REGION Network 115: NG 1 Door NOT Closed
   RUNG wire#powerrail
      Contact( "AlwaysTRUE" )
      Contact( "Station_Sys".Auto.Mode )
      I_Contact( "oE-NG-01SafetyGate" )
      Coil( "ST10_DeviceError"."E".NG_1."NG 1 DoorOpen" )
   END_RUNG
   // the same network as SCL:
   "ST10_DeviceError"."E".NG_1."NG 1 DoorOpen" := "AlwaysTRUE" AND "Station_Sys".Auto.Mode AND NOT "oE-NG-01SafetyGate";
END_REGION

REGION Network 116: E NG_2
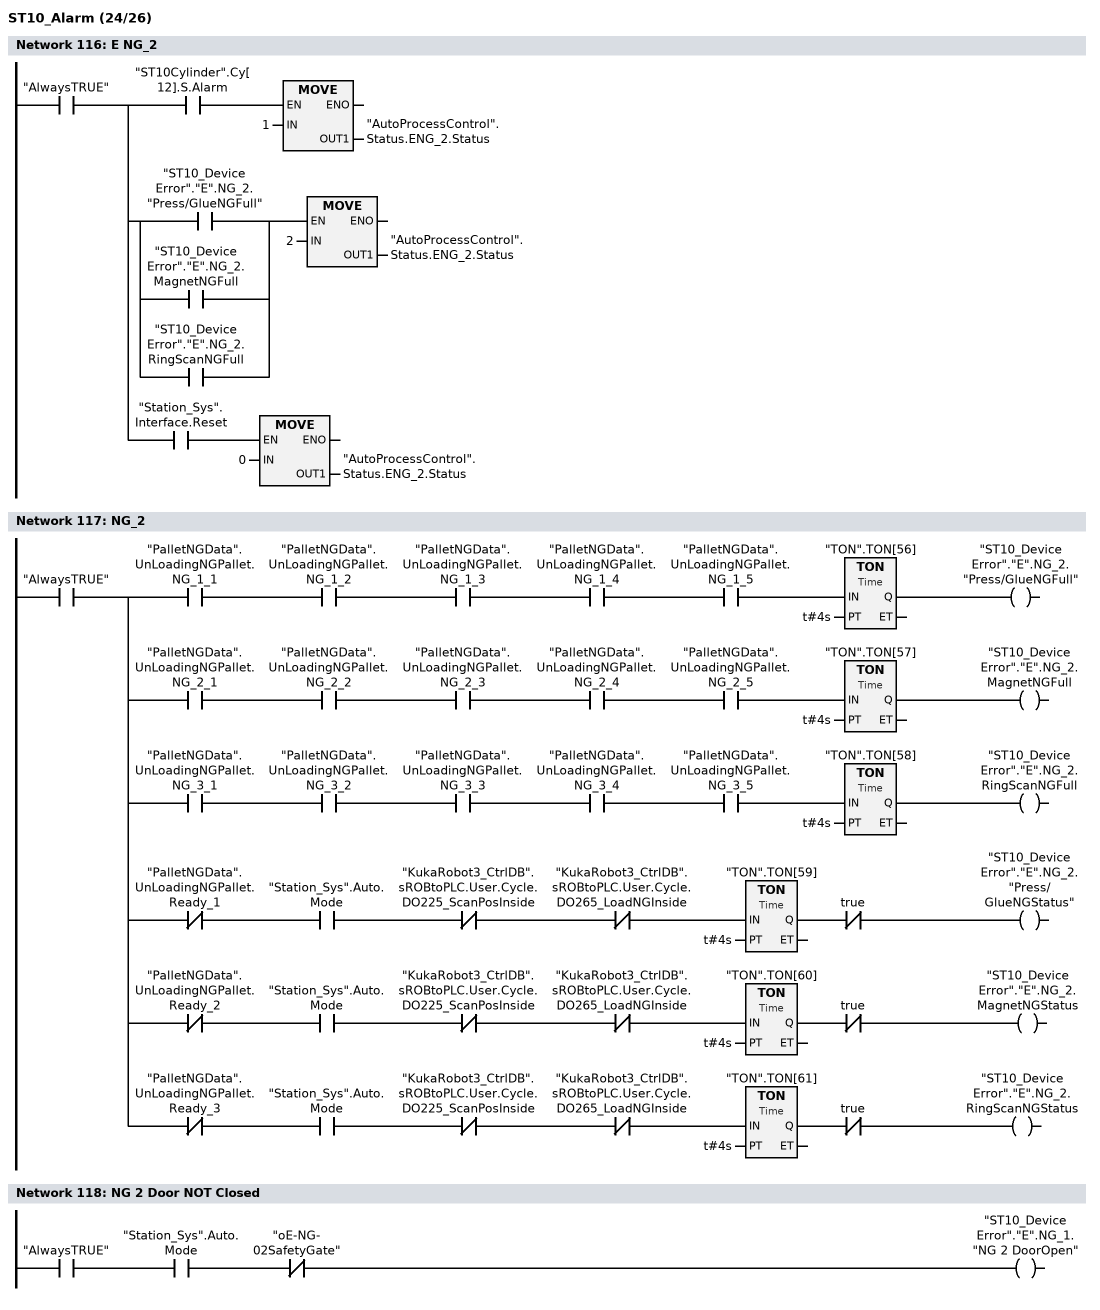
   RUNG wire#powerrail
      Contact( "AlwaysTRUE" )
      wire#w1
      Contact( "ST10Cylinder".Cy[12].S.Alarm )
      Move(in := 1, out1 => "AutoProcessControl".Status.ENG_2.Status)
   END_RUNG
   RUNG wire#w1
      Contact( "ST10_DeviceError"."E".NG_2."Press/GlueNGFull" )
      wire#w2
      Move(in := 2, out1 => "AutoProcessControl".Status.ENG_2.Status)
   END_RUNG
   RUNG wire#w1
      Contact( "ST10_DeviceError"."E".NG_2.MagnetNGFull )
   END_RUNG wire#w2
   RUNG wire#w1
      Contact( "ST10_DeviceError"."E".NG_2.RingScanNGFull )
   END_RUNG wire#w2
   RUNG wire#w1
      Contact( "Station_Sys".Interface.Reset )
      Move(in := 0, out1 => "AutoProcessControl".Status.ENG_2.Status)
   END_RUNG
   // the same network as SCL:
   IF "AlwaysTRUE" AND "ST10Cylinder".Cy[12].S.Alarm THEN
       "AutoProcessControl".Status.ENG_2.Status := 1;
   END_IF;
   IF "AlwaysTRUE" AND ("ST10_DeviceError"."E".NG_2."Press/GlueNGFull" OR "ST10_DeviceError"."E".NG_2.MagnetNGFull OR "ST10_DeviceError"."E".NG_2.RingScanNGFull) THEN
       "AutoProcessControl".Status.ENG_2.Status := 2;
   END_IF;
   IF "AlwaysTRUE" AND "Station_Sys".Interface.Reset THEN
       "AutoProcessControl".Status.ENG_2.Status := 0;
   END_IF;
END_REGION

REGION Network 117: NG_2
   RUNG wire#powerrail
      Contact( "AlwaysTRUE" )
      wire#w1
      Contact( "PalletNGData".UnLoadingNGPallet.NG_1_1 )
      Contact( "PalletNGData".UnLoadingNGPallet.NG_1_2 )
      Contact( "PalletNGData".UnLoadingNGPallet.NG_1_3 )
      Contact( "PalletNGData".UnLoadingNGPallet.NG_1_4 )
      Contact( "PalletNGData".UnLoadingNGPallet.NG_1_5 )
      { S7_Templates := "time_type := Time" } "TON".TON[56].TON(pt := t#4s, et =>)
      Coil( "ST10_DeviceError"."E".NG_2."Press/GlueNGFull" )
   END_RUNG
   RUNG wire#w1
      Contact( "PalletNGData".UnLoadingNGPallet.NG_2_1 )
      Contact( "PalletNGData".UnLoadingNGPallet.NG_2_2 )
      Contact( "PalletNGData".UnLoadingNGPallet.NG_2_3 )
      Contact( "PalletNGData".UnLoadingNGPallet.NG_2_4 )
      Contact( "PalletNGData".UnLoadingNGPallet.NG_2_5 )
      { S7_Templates := "time_type := Time" } "TON".TON[57].TON(pt := t#4s, et =>)
      Coil( "ST10_DeviceError"."E".NG_2.MagnetNGFull )
   END_RUNG
   RUNG wire#w1
      Contact( "PalletNGData".UnLoadingNGPallet.NG_3_1 )
      Contact( "PalletNGData".UnLoadingNGPallet.NG_3_2 )
      Contact( "PalletNGData".UnLoadingNGPallet.NG_3_3 )
      Contact( "PalletNGData".UnLoadingNGPallet.NG_3_4 )
      Contact( "PalletNGData".UnLoadingNGPallet.NG_3_5 )
      { S7_Templates := "time_type := Time" } "TON".TON[58].TON(pt := t#4s, et =>)
      Coil( "ST10_DeviceError"."E".NG_2.RingScanNGFull )
   END_RUNG
   RUNG wire#w1
      I_Contact( "PalletNGData".UnLoadingNGPallet.Ready_1 )
      Contact( "Station_Sys".Auto.Mode )
      I_Contact( "KukaRobot3_CtrlDB".sROBtoPLC.User.Cycle.DO225_ScanPosInside )
      I_Contact( "KukaRobot3_CtrlDB".sROBtoPLC.User.Cycle.DO265_LoadNGInside )
      { S7_Templates := "time_type := Time" } "TON".TON[59].TON(pt := t#4s, et =>)
      I_Contact( true )
      Coil( "ST10_DeviceError"."E".NG_2."Press/GlueNGStatus" )
   END_RUNG
   RUNG wire#w1
      I_Contact( "PalletNGData".UnLoadingNGPallet.Ready_2 )
      Contact( "Station_Sys".Auto.Mode )
      I_Contact( "KukaRobot3_CtrlDB".sROBtoPLC.User.Cycle.DO225_ScanPosInside )
      I_Contact( "KukaRobot3_CtrlDB".sROBtoPLC.User.Cycle.DO265_LoadNGInside )
      { S7_Templates := "time_type := Time" } "TON".TON[60].TON(pt := t#4s, et =>)
      I_Contact( true )
      Coil( "ST10_DeviceError"."E".NG_2.MagnetNGStatus )
   END_RUNG
   RUNG wire#w1
      I_Contact( "PalletNGData".UnLoadingNGPallet.Ready_3 )
      Contact( "Station_Sys".Auto.Mode )
      I_Contact( "KukaRobot3_CtrlDB".sROBtoPLC.User.Cycle.DO225_ScanPosInside )
      I_Contact( "KukaRobot3_CtrlDB".sROBtoPLC.User.Cycle.DO265_LoadNGInside )
      { S7_Templates := "time_type := Time" } "TON".TON[61].TON(pt := t#4s, et =>)
      I_Contact( true )
      Coil( "ST10_DeviceError"."E".NG_2.RingScanNGStatus )
   END_RUNG
   // the same network as SCL:
   "TON".TON[56].TON(IN := "AlwaysTRUE" AND "PalletNGData".UnLoadingNGPallet.NG_1_1 AND "PalletNGData".UnLoadingNGPallet.NG_1_2 AND "PalletNGData".UnLoadingNGPallet.NG_1_3 AND "PalletNGData".UnLoadingNGPallet.NG_1_4 AND "PalletNGData".UnLoadingNGPallet.NG_1_5,
                     PT := t#4s);
   "ST10_DeviceError"."E".NG_2."Press/GlueNGFull" := "TON".TON[56].Q;
   "TON".TON[57].TON(IN := "AlwaysTRUE" AND "PalletNGData".UnLoadingNGPallet.NG_2_1 AND "PalletNGData".UnLoadingNGPallet.NG_2_2 AND "PalletNGData".UnLoadingNGPallet.NG_2_3 AND "PalletNGData".UnLoadingNGPallet.NG_2_4 AND "PalletNGData".UnLoadingNGPallet.NG_2_5,
                     PT := t#4s);
   "ST10_DeviceError"."E".NG_2.MagnetNGFull := "TON".TON[57].Q;
   "TON".TON[58].TON(IN := "AlwaysTRUE" AND "PalletNGData".UnLoadingNGPallet.NG_3_1 AND "PalletNGData".UnLoadingNGPallet.NG_3_2 AND "PalletNGData".UnLoadingNGPallet.NG_3_3 AND "PalletNGData".UnLoadingNGPallet.NG_3_4 AND "PalletNGData".UnLoadingNGPallet.NG_3_5,
                     PT := t#4s);
   "ST10_DeviceError"."E".NG_2.RingScanNGFull := "TON".TON[58].Q;
   "TON".TON[59].TON(IN := "AlwaysTRUE" AND NOT "PalletNGData".UnLoadingNGPallet.Ready_1 AND "Station_Sys".Auto.Mode AND NOT "KukaRobot3_CtrlDB".sROBtoPLC.User.Cycle.DO225_ScanPosInside AND NOT "KukaRobot3_CtrlDB".sROBtoPLC.User.Cycle.DO265_LoadNGInside,
                     PT := t#4s);
   "ST10_DeviceError"."E".NG_2."Press/GlueNGStatus" := "TON".TON[59].Q AND NOT true;
   "TON".TON[60].TON(IN := "AlwaysTRUE" AND NOT "PalletNGData".UnLoadingNGPallet.Ready_2 AND "Station_Sys".Auto.Mode AND NOT "KukaRobot3_CtrlDB".sROBtoPLC.User.Cycle.DO225_ScanPosInside AND NOT "KukaRobot3_CtrlDB".sROBtoPLC.User.Cycle.DO265_LoadNGInside,
                     PT := t#4s);
   "ST10_DeviceError"."E".NG_2.MagnetNGStatus := "TON".TON[60].Q AND NOT true;
   "TON".TON[61].TON(IN := "AlwaysTRUE" AND NOT "PalletNGData".UnLoadingNGPallet.Ready_3 AND "Station_Sys".Auto.Mode AND NOT "KukaRobot3_CtrlDB".sROBtoPLC.User.Cycle.DO225_ScanPosInside AND NOT "KukaRobot3_CtrlDB".sROBtoPLC.User.Cycle.DO265_LoadNGInside,
                     PT := t#4s);
   "ST10_DeviceError"."E".NG_2.RingScanNGStatus := "TON".TON[61].Q AND NOT true;
END_REGION

REGION Network 118: NG 2 Door NOT Closed
   RUNG wire#powerrail
      Contact( "AlwaysTRUE" )
      Contact( "Station_Sys".Auto.Mode )
      I_Contact( "oE-NG-02SafetyGate" )
      Coil( "ST10_DeviceError"."E".NG_1."NG 2 DoorOpen" )
   END_RUNG
   // the same network as SCL:
   "ST10_DeviceError"."E".NG_1."NG 2 DoorOpen" := "AlwaysTRUE" AND "Station_Sys".Auto.Mode AND NOT "oE-NG-02SafetyGate";
END_REGION

REGION Network 119: Press1
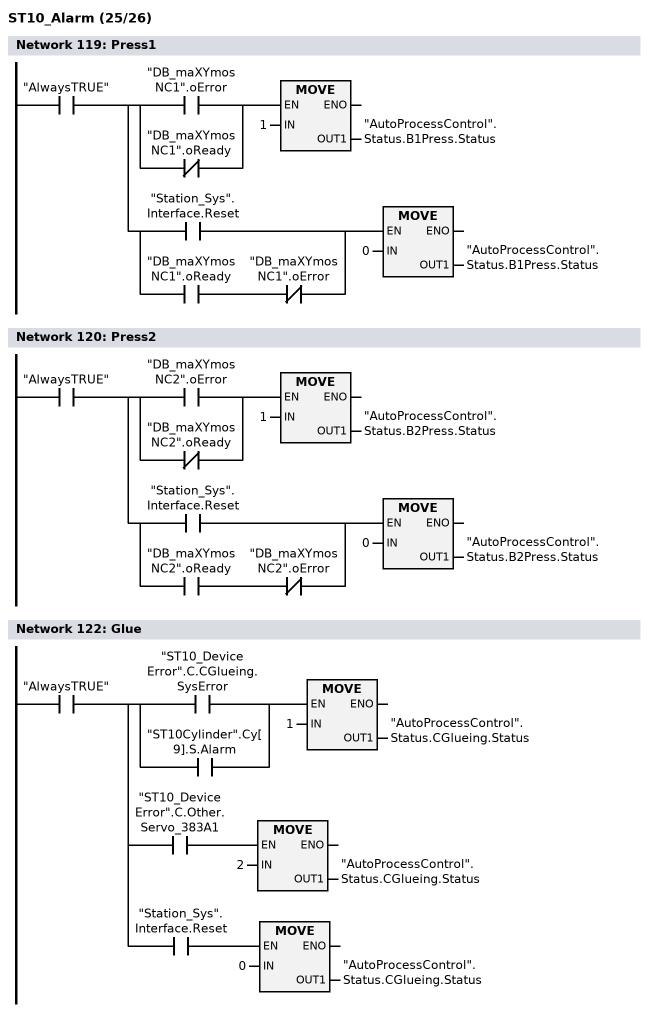
   RUNG wire#powerrail
      Contact( "AlwaysTRUE" )
      wire#w1
      Contact( "DB_maXYmosNC1".oError )
      wire#w2
      Move(in := 1, out1 => "AutoProcessControl".Status.B1Press.Status)
   END_RUNG
   RUNG wire#w1
      I_Contact( "DB_maXYmosNC1".oReady )
   END_RUNG wire#w2
   RUNG wire#w1
      Contact( "Station_Sys".Interface.Reset )
      wire#w3
      Move(in := 0, out1 => "AutoProcessControl".Status.B1Press.Status)
   END_RUNG
   RUNG wire#w1
      Contact( "DB_maXYmosNC1".oReady )
      I_Contact( "DB_maXYmosNC1".oError )
   END_RUNG wire#w3
   // the same network as SCL:
   IF "AlwaysTRUE" AND ("DB_maXYmosNC1".oError OR NOT "DB_maXYmosNC1".oReady) THEN
       "AutoProcessControl".Status.B1Press.Status := 1;
   END_IF;
   IF "AlwaysTRUE" AND ("Station_Sys".Interface.Reset OR ("DB_maXYmosNC1".oReady AND NOT "DB_maXYmosNC1".oError)) THEN
       "AutoProcessControl".Status.B1Press.Status := 0;
   END_IF;
END_REGION

REGION Network 120: Press2
   RUNG wire#powerrail
      Contact( "AlwaysTRUE" )
      wire#w1
      Contact( "DB_maXYmosNC2".oError )
      wire#w2
      Move(in := 1, out1 => "AutoProcessControl".Status.B2Press.Status)
   END_RUNG
   RUNG wire#w1
      I_Contact( "DB_maXYmosNC2".oReady )
   END_RUNG wire#w2
   RUNG wire#w1
      Contact( "Station_Sys".Interface.Reset )
      wire#w3
      Move(in := 0, out1 => "AutoProcessControl".Status.B2Press.Status)
   END_RUNG
   RUNG wire#w1
      Contact( "DB_maXYmosNC2".oReady )
      I_Contact( "DB_maXYmosNC2".oError )
   END_RUNG wire#w3
   // the same network as SCL:
   IF "AlwaysTRUE" AND ("DB_maXYmosNC2".oError OR NOT "DB_maXYmosNC2".oReady) THEN
       "AutoProcessControl".Status.B2Press.Status := 1;
   END_IF;
   IF "AlwaysTRUE" AND ("Station_Sys".Interface.Reset OR ("DB_maXYmosNC2".oReady AND NOT "DB_maXYmosNC2".oError)) THEN
       "AutoProcessControl".Status.B2Press.Status := 0;
   END_IF;
END_REGION

REGION Network 121: ******************** Glue ********************
END_REGION

REGION Network 122: Glue
   RUNG wire#powerrail
      Contact( "AlwaysTRUE" )
      wire#w1
      Contact( "ST10_DeviceError".C.CGlueing.SysError )
      wire#w2
      Move(in := 1, out1 => "AutoProcessControl".Status.CGlueing.Status)
   END_RUNG
   RUNG wire#w1
      Contact( "ST10Cylinder".Cy[9].S.Alarm )
   END_RUNG wire#w2
   RUNG wire#w1
      Contact( "ST10_DeviceError".C.Other.Servo_383A1 )
      Move(in := 2, out1 => "AutoProcessControl".Status.CGlueing.Status)
   END_RUNG
   RUNG wire#w1
      Contact( "Station_Sys".Interface.Reset )
      Move(in := 0, out1 => "AutoProcessControl".Status.CGlueing.Status)
   END_RUNG
   // the same network as SCL:
   IF "AlwaysTRUE" AND ("ST10_DeviceError".C.CGlueing.SysError OR "ST10Cylinder".Cy[9].S.Alarm) THEN
       "AutoProcessControl".Status.CGlueing.Status := 1;
   END_IF;
   IF "AlwaysTRUE" AND "ST10_DeviceError".C.Other.Servo_383A1 THEN
       "AutoProcessControl".Status.CGlueing.Status := 2;
   END_IF;
   IF "AlwaysTRUE" AND "Station_Sys".Interface.Reset THEN
       "AutoProcessControl".Status.CGlueing.Status := 0;
   END_IF;
END_REGION

REGION Network 123: A1 Table
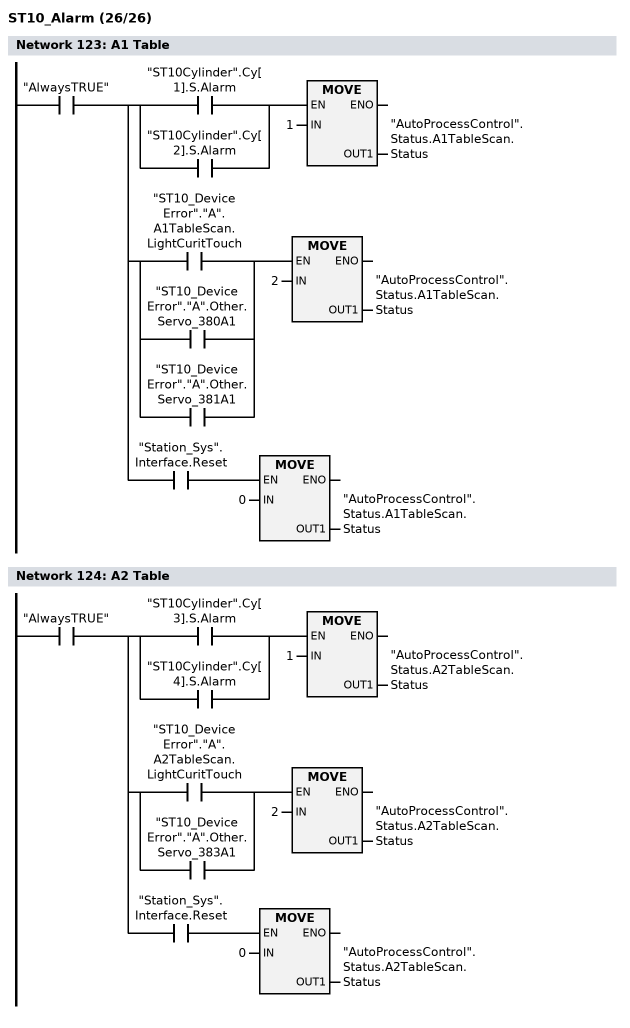
   RUNG wire#powerrail
      Contact( "AlwaysTRUE" )
      wire#w1
      Contact( "ST10Cylinder".Cy[1].S.Alarm )
      wire#w2
      Move(in := 1, out1 => "AutoProcessControl".Status.A1TableScan.Status)
   END_RUNG
   RUNG wire#w1
      Contact( "ST10Cylinder".Cy[2].S.Alarm )
   END_RUNG wire#w2
   RUNG wire#w1
      Contact( "ST10_DeviceError"."A".A1TableScan.LightCuritTouch )
      wire#w3
      Move(in := 2, out1 => "AutoProcessControl".Status.A1TableScan.Status)
   END_RUNG
   RUNG wire#w1
      Contact( "ST10_DeviceError"."A".Other.Servo_380A1 )
   END_RUNG wire#w3
   RUNG wire#w1
      Contact( "ST10_DeviceError"."A".Other.Servo_381A1 )
   END_RUNG wire#w3
   RUNG wire#w1
      Contact( "Station_Sys".Interface.Reset )
      Move(in := 0, out1 => "AutoProcessControl".Status.A1TableScan.Status)
   END_RUNG
   // the same network as SCL:
   IF "AlwaysTRUE" AND ("ST10Cylinder".Cy[1].S.Alarm OR "ST10Cylinder".Cy[2].S.Alarm) THEN
       "AutoProcessControl".Status.A1TableScan.Status := 1;
   END_IF;
   IF "AlwaysTRUE" AND ("ST10_DeviceError"."A".A1TableScan.LightCuritTouch OR "ST10_DeviceError"."A".Other.Servo_380A1 OR "ST10_DeviceError"."A".Other.Servo_381A1) THEN
       "AutoProcessControl".Status.A1TableScan.Status := 2;
   END_IF;
   IF "AlwaysTRUE" AND "Station_Sys".Interface.Reset THEN
       "AutoProcessControl".Status.A1TableScan.Status := 0;
   END_IF;
END_REGION

REGION Network 124: A2 Table
   RUNG wire#powerrail
      Contact( "AlwaysTRUE" )
      wire#w1
      Contact( "ST10Cylinder".Cy[3].S.Alarm )
      wire#w2
      Move(in := 1, out1 => "AutoProcessControl".Status.A2TableScan.Status)
   END_RUNG
   RUNG wire#w1
      Contact( "ST10Cylinder".Cy[4].S.Alarm )
   END_RUNG wire#w2
   RUNG wire#w1
      Contact( "ST10_DeviceError"."A".A2TableScan.LightCuritTouch )
      wire#w3
      Move(in := 2, out1 => "AutoProcessControl".Status.A2TableScan.Status)
   END_RUNG
   RUNG wire#w1
      Contact( "ST10_DeviceError"."A".Other.Servo_383A1 )
   END_RUNG wire#w3
   RUNG wire#w1
      Contact( "Station_Sys".Interface.Reset )
      Move(in := 0, out1 => "AutoProcessControl".Status.A2TableScan.Status)
   END_RUNG
   // the same network as SCL:
   IF "AlwaysTRUE" AND ("ST10Cylinder".Cy[3].S.Alarm OR "ST10Cylinder".Cy[4].S.Alarm) THEN
       "AutoProcessControl".Status.A2TableScan.Status := 1;
   END_IF;
   IF "AlwaysTRUE" AND ("ST10_DeviceError"."A".A2TableScan.LightCuritTouch OR "ST10_DeviceError"."A".Other.Servo_383A1) THEN
       "AutoProcessControl".Status.A2TableScan.Status := 2;
   END_IF;
   IF "AlwaysTRUE" AND "Station_Sys".Interface.Reset THEN
       "AutoProcessControl".Status.A2TableScan.Status := 0;
   END_IF;
END_REGION
END_FUNCTION

FUNCTION "ST10Cyl_interface11-20" : Void   // FC1021, LAD
{ S7_Optimized_Access := 'FALSE' }
// stored: AutoNumber false, SetENOAutomatically false
   VAR_INPUT
      AlwaysON : Bool;
      E_stop : Bool;
   END_VAR
   VAR_TEMP
      tTest : Bool;
   END_VAR
BEGIN

REGION Network 1 (SCL): Cylinder 11-20 IO Interface (SCL)

   //Cylinder11 IO   E-NG-01NGLocationCylinder
   //Input
   "ST10Cylinder".Cy[11].In.WorkPositionSensor := "iE-NG-01NGLocationCylinderInWP";
   "ST10Cylinder".Cy[11].In.HomePositionSensor := "iE-NG-01NGLocationCylinderInHP";
   //Output
   "oE-NG-01NGLocationCylinderToWP" := "ST10Cylinder".Cy[11].Out.GoWorkPosition;
   "oE-NG-01NGLocationCylinderToHP" := "ST10Cylinder".Cy[11].Out.GoHomePosition;

   //Cylinder12 IO  E-NG-02NGLocationCylinder
   //Input
   "ST10Cylinder".Cy[12].In.WorkPositionSensor := "iE-NG-02NGLocationCylinderInWP";
   "ST10Cylinder".Cy[12].In.HomePositionSensor := "iE-NG-02NGLocationCylinderInHP";
   //Output
   "oE-NG-02NGLocationCylinderToWP" := "ST10Cylinder".Cy[12].Out.GoWorkPosition;
   "oE-NG-02NGLocationCylinderToHP" := "ST10Cylinder".Cy[12].Out.GoHomePosition;

   //Cylinder13 IO  F-ROOBT1Gripper1Cylinder
   //Input
   "KukaRobot1_CtrlDB".sPLCtoROB.User.Gripper.DI129_Grip1WP:="ST10Cylinder".Cy[13].In.WorkPositionSensor := "iF-ROOBT1Gripper1CylinderInWP" ;
   "KukaRobot1_CtrlDB".sPLCtoROB.User.Gripper.DI130_Grip1HP := "ST10Cylinder".Cy[13].In.HomePositionSensor := "iF-ROOBT1Gripper1CylinderInHP" ;//"TON".TON[0].Q;

   IF  NOT "Robot_DB".Control.Robot1GripControl THEN
       //Output
       "oF-ROOBT1Gripper1CylinderToWP" := "KukaRobot1_CtrlDB".sROBtoPLC.User.Gripper.DO129_Grip1GoWork;
       "oF-ROOBT1Gripper1CylinderToHP" := "KukaRobot1_CtrlDB".sROBtoPLC.User.Gripper.DO130_Grip1GoHome;
   ELSE
       //Output
       "oF-ROOBT1Gripper1CylinderToWP" := "ST10Cylinder".Cy[13].Out.GoWorkPosition;
       "oF-ROOBT1Gripper1CylinderToHP" := "ST10Cylinder".Cy[13].Out.GoHomePosition;
   END_IF;
   "TON".TON[0](IN:="oF-ROOBT1Gripper1CylinderToHP" AND NOT"iF-ROOBT1Gripper1CylinderInWP",PT:=T#500MS);


   //Cylinder14 IO  F-ROOBT1Gripper2Cylinder
   //Input
   "KukaRobot1_CtrlDB".sPLCtoROB.User.Gripper.DI131_Grip2WP:="ST10Cylinder".Cy[14].In.WorkPositionSensor := "iF-ROOBT1Gripper2CylinderInWP";
   "KukaRobot1_CtrlDB".sPLCtoROB.User.Gripper.DI132_Grip2HP:="ST10Cylinder".Cy[14].In.HomePositionSensor := "iF-ROOBT1Gripper2CylinderInHP";

   IF NOT "Robot_DB".Control.Robot1GripControl THEN
       //Output
       "oF-ROOBT1Gripper2CylinderToWP" :="ST10Cylinder".Cy[14].Inout.AutoGoWork:="KukaRobot1_CtrlDB".sROBtoPLC.User.Gripper.DO131_Grip2GoWork;
       "oF-ROOBT1Gripper2CylinderToHP" :="ST10Cylinder".Cy[14].Inout.AutoGoHome:="KukaRobot1_CtrlDB".sROBtoPLC.User.Gripper.DO132_Grip2GoHome;
   ELSE
       //Output
       "oF-ROOBT1Gripper2CylinderToWP" := "ST10Cylinder".Cy[14].Out.GoWorkPosition;
       "oF-ROOBT1Gripper2CylinderToHP" := "ST10Cylinder".Cy[14].Out.GoHomePosition;
   END_IF;


   //Cylinder15 IO  F-ROOBT2Gripper1Cylinder
   //Input
   "KukaRobot2_CtrlDB".sPLCtoROB.User.Gripper.DI129_Grip1WP:="ST10Cylinder".Cy[15].In.WorkPositionSensor := "iF-ROOBT2Gripper1CylinderInWP";
   "KukaRobot2_CtrlDB".sPLCtoROB.User.Gripper.DI130_Grip1HP := "ST10Cylinder".Cy[15].In.HomePositionSensor :="iF-ROOBT2Gripper1CylinderInHP";

   IF NOT "Robot_DB".Control.Robot2GripControl THEN
       //Output
       "oF-ROOBT2Gripper1CylinderToWP" :="ST10Cylinder".Cy[15].Inout.AutoGoWork:="KukaRobot2_CtrlDB".sROBtoPLC.User.Gripper.DO129_Grip1GoWork;
       "oF-ROOBT2Gripper1CylinderToHP" :="ST10Cylinder".Cy[15].Inout.AutoGoHome:="KukaRobot2_CtrlDB".sROBtoPLC.User.Gripper.DO130_Grip1GoHome;
   ELSE
       //Output
       "oF-ROOBT2Gripper1CylinderToWP" := "ST10Cylinder".Cy[15].Out.GoWorkPosition;
       "oF-ROOBT2Gripper1CylinderToHP" := "ST10Cylinder".Cy[15].Out.GoHomePosition;
   END_IF;



   //Cylinder16 IO  F-ROOBT2Gripper2Cylinder
   //Input
   "KukaRobot2_CtrlDB".sPLCtoROB.User.Gripper.DI131_Grip2WP:="ST10Cylinder".Cy[16].In.WorkPositionSensor := "iF-ROOBT2Gripper2CylinderInWP";
   "KukaRobot2_CtrlDB".sPLCtoROB.User.Gripper.DI132_Grip2HP:="ST10Cylinder".Cy[16].In.HomePositionSensor := "iF-ROOBT2Gripper2CylinderInHP";

   IF NOT "Robot_DB".Control.Robot2GripControl THEN
       //Output
       "oF-ROOBT2Gripper2CylinderToWP" :="ST10Cylinder".Cy[16].Inout.AutoGoWork:= "KukaRobot2_CtrlDB".sROBtoPLC.User.Gripper.DO131_Grip2GoWork;
       "oF-ROOBT2Gripper2CylinderToHP" :="ST10Cylinder".Cy[16].Inout.AutoGoHome:= "KukaRobot2_CtrlDB".sROBtoPLC.User.Gripper.DO132_Grip2GoHome;
   ELSE
       //Output
       "oF-ROOBT2Gripper2CylinderToWP" := "ST10Cylinder".Cy[16].Out.GoWorkPosition;
       "oF-ROOBT2Gripper2CylinderToHP" := "ST10Cylinder".Cy[16].Out.GoHomePosition;
   END_IF;

   //Cylinder17 IO  F-ROOBT3Gripper1Cylinder
   //Input
   "KukaRobot3_CtrlDB".sPLCtoROB.User.Gripper.DI129_Grip1WP:="ST10Cylinder".Cy[17].In.WorkPositionSensor := "iF-ROOBT3Gripper1CylinderInWP";
   "KukaRobot3_CtrlDB".sPLCtoROB.User.Gripper.DI130_Grip1HP:="ST10Cylinder".Cy[17].In.HomePositionSensor := "iF-ROOBT3Gripper1CylinderInHP";

   IF NOT "Robot_DB".Control.Robot3GripControl THEN
       //Output
       "oF-ROOBT3Gripper1CylinderToWP" :="ST10Cylinder".Cy[17].Inout.AutoGoWork:="KukaRobot3_CtrlDB".sROBtoPLC.User.Gripper.DO129_Grip1GoWork;
       "oF-ROOBT3Gripper1CylinderToHP" :="ST10Cylinder".Cy[17].Inout.AutoGoHome:="KukaRobot3_CtrlDB".sROBtoPLC.User.Gripper.DO130_Grip1GoHome;
   ELSE
       //Output
       "oF-ROOBT3Gripper1CylinderToWP" := "ST10Cylinder".Cy[17].Out.GoWorkPosition;
       "oF-ROOBT3Gripper1CylinderToHP" := "ST10Cylinder".Cy[17].Out.GoHomePosition;
   END_IF;


   //Cylinder18 IO  F-ROOBT3Gripper2Cylinder
   //Input
   "KukaRobot3_CtrlDB".sPLCtoROB.User.Gripper.DI131_Grip2WP:="ST10Cylinder".Cy[18].In.WorkPositionSensor := "iF-ROOBT3Gripper2CylinderInWP";
   "KukaRobot3_CtrlDB".sPLCtoROB.User.Gripper.DI132_Grip2HP := "ST10Cylinder".Cy[18].In.HomePositionSensor := "iF-ROOBT3Gripper2CylinderInHP";//"TON".TON[1].Q;

   IF NOT "Robot_DB".Control.Robot3GripControl THEN
       //Output
       "oF-ROOBT3Gripper2CylinderToWP" :="ST10Cylinder".Cy[18].Inout.AutoGoWork:="KukaRobot3_CtrlDB".sROBtoPLC.User.Gripper.DO131_Grip2GoWork;
       "oF-ROOBT3Gripper2CylinderToHP" :="ST10Cylinder".Cy[18].Inout.AutoGoHome:="KukaRobot3_CtrlDB".sROBtoPLC.User.Gripper.DO132_Grip2GoHome;
   ELSE
       //Output
       "oF-ROOBT3Gripper2CylinderToWP" := "ST10Cylinder".Cy[18].Out.GoWorkPosition;
       "oF-ROOBT3Gripper2CylinderToHP" := "ST10Cylinder".Cy[18].Out.GoHomePosition;
   END_IF;

   "TON".TON[1](IN := "oF-ROOBT3Gripper2CylinderToHP" AND NOT "iF-ROOBT3Gripper2CylinderInWP",
                PT := T#500MS);

   (*
   //Cylinder19 IO  D-washer Loading Horizontal
   //Input
   "ST10Cylinder".Cy[19].In.WorkPositionSensor := ("D-washer Loading Cylinder Middle Cylinder InHP" AND "D-washer Loading Horizontal Cylinder InWP")
                                               OR ("D-washer Loading Cylinder Middle Cylinder InWP" AND "D-washer Loading Horizontal Cylinder InWP1");
   "ST10Cylinder".Cy[19].In.HomePositionSensor := "D-washer Loading Horizontal Cylinder InHP";
   //Output
   "D-washer Loading Horizontal Cylinder ToWP" := "ST10Cylinder".Cy[19].Out.GoWorkPosition;
   "D-washer Loading Horizontal Cylinder ToHP" := "ST10Cylinder".Cy[19].Out.GoHomePosition;

   //Cylinder20 IO  D-washer Loading Cylinder Middle
   //Input
   "ST10Cylinder".Cy[20].In.WorkPositionSensor := "D-washer Loading Cylinder Middle Cylinder InWP";
   "ST10Cylinder".Cy[20].In.HomePositionSensor := "D-washer Loading Cylinder Middle Cylinder InHP";
   //Output
   "D-washer Loading Cylinder Middle Cylinder ToWP" := "ST10Cylinder".Cy[20].Out.GoWorkPosition;
   "D-washer Loading Cylinder Middle Cylinder ToHP" := "ST10Cylinder".Cy[20].Out.GoHomePosition;
   *)
END_REGION

REGION Network 2: CY11 interface E-NG-01NGLocationCylinder
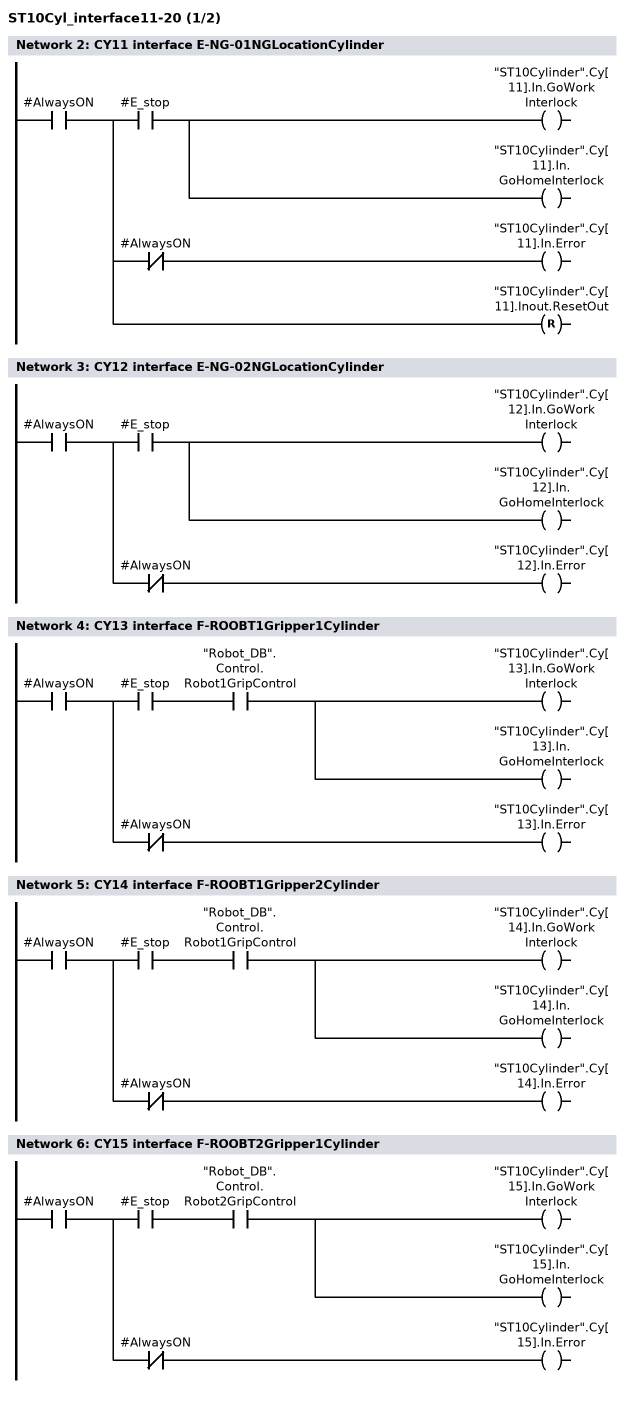
   RUNG wire#powerrail
      Contact( #AlwaysON )
      wire#w1
      Contact( #E_stop )
      wire#w2
      Coil( "ST10Cylinder".Cy[11].In.GoWorkInterlock )
   END_RUNG
   RUNG wire#w2
      Coil( "ST10Cylinder".Cy[11].In.GoHomeInterlock )
   END_RUNG
   RUNG wire#w1
      I_Contact( #AlwaysON )
      Coil( "ST10Cylinder".Cy[11].In.Error )
   END_RUNG
   RUNG wire#w1
      R_Coil( "ST10Cylinder".Cy[11].Inout.ResetOut )
   END_RUNG
   // the same network as SCL:
   "ST10Cylinder".Cy[11].In.GoWorkInterlock := #AlwaysON AND #E_stop;
   "ST10Cylinder".Cy[11].In.GoHomeInterlock := #AlwaysON AND #E_stop;
   "ST10Cylinder".Cy[11].In.Error := #AlwaysON AND NOT #AlwaysON;
   IF #AlwaysON THEN "ST10Cylinder".Cy[11].Inout.ResetOut := FALSE; END_IF;
END_REGION

REGION Network 3: CY12 interface E-NG-02NGLocationCylinder
   RUNG wire#powerrail
      Contact( #AlwaysON )
      wire#w1
      Contact( #E_stop )
      wire#w2
      Coil( "ST10Cylinder".Cy[12].In.GoWorkInterlock )
   END_RUNG
   RUNG wire#w2
      Coil( "ST10Cylinder".Cy[12].In.GoHomeInterlock )
   END_RUNG
   RUNG wire#w1
      I_Contact( #AlwaysON )
      Coil( "ST10Cylinder".Cy[12].In.Error )
   END_RUNG
   // the same network as SCL:
   "ST10Cylinder".Cy[12].In.GoWorkInterlock := #AlwaysON AND #E_stop;
   "ST10Cylinder".Cy[12].In.GoHomeInterlock := #AlwaysON AND #E_stop;
   "ST10Cylinder".Cy[12].In.Error := #AlwaysON AND NOT #AlwaysON;
END_REGION

REGION Network 4: CY13 interface F-ROOBT1Gripper1Cylinder
   RUNG wire#powerrail
      Contact( #AlwaysON )
      wire#w1
      Contact( #E_stop )
      Contact( "Robot_DB".Control.Robot1GripControl )
      wire#w2
      Coil( "ST10Cylinder".Cy[13].In.GoWorkInterlock )
   END_RUNG
   RUNG wire#w2
      Coil( "ST10Cylinder".Cy[13].In.GoHomeInterlock )
   END_RUNG
   RUNG wire#w1
      I_Contact( #AlwaysON )
      Coil( "ST10Cylinder".Cy[13].In.Error )
   END_RUNG
   // the same network as SCL:
   "ST10Cylinder".Cy[13].In.GoWorkInterlock := #AlwaysON AND #E_stop AND "Robot_DB".Control.Robot1GripControl;
   "ST10Cylinder".Cy[13].In.GoHomeInterlock := #AlwaysON AND #E_stop AND "Robot_DB".Control.Robot1GripControl;
   "ST10Cylinder".Cy[13].In.Error := #AlwaysON AND NOT #AlwaysON;
END_REGION

REGION Network 5: CY14 interface F-ROOBT1Gripper2Cylinder
   RUNG wire#powerrail
      Contact( #AlwaysON )
      wire#w1
      Contact( #E_stop )
      Contact( "Robot_DB".Control.Robot1GripControl )
      wire#w2
      Coil( "ST10Cylinder".Cy[14].In.GoWorkInterlock )
   END_RUNG
   RUNG wire#w2
      Coil( "ST10Cylinder".Cy[14].In.GoHomeInterlock )
   END_RUNG
   RUNG wire#w1
      I_Contact( #AlwaysON )
      Coil( "ST10Cylinder".Cy[14].In.Error )
   END_RUNG
   // the same network as SCL:
   "ST10Cylinder".Cy[14].In.GoWorkInterlock := #AlwaysON AND #E_stop AND "Robot_DB".Control.Robot1GripControl;
   "ST10Cylinder".Cy[14].In.GoHomeInterlock := #AlwaysON AND #E_stop AND "Robot_DB".Control.Robot1GripControl;
   "ST10Cylinder".Cy[14].In.Error := #AlwaysON AND NOT #AlwaysON;
END_REGION

REGION Network 6: CY15 interface F-ROOBT2Gripper1Cylinder
   RUNG wire#powerrail
      Contact( #AlwaysON )
      wire#w1
      Contact( #E_stop )
      Contact( "Robot_DB".Control.Robot2GripControl )
      wire#w2
      Coil( "ST10Cylinder".Cy[15].In.GoWorkInterlock )
   END_RUNG
   RUNG wire#w2
      Coil( "ST10Cylinder".Cy[15].In.GoHomeInterlock )
   END_RUNG
   RUNG wire#w1
      I_Contact( #AlwaysON )
      Coil( "ST10Cylinder".Cy[15].In.Error )
   END_RUNG
   // the same network as SCL:
   "ST10Cylinder".Cy[15].In.GoWorkInterlock := #AlwaysON AND #E_stop AND "Robot_DB".Control.Robot2GripControl;
   "ST10Cylinder".Cy[15].In.GoHomeInterlock := #AlwaysON AND #E_stop AND "Robot_DB".Control.Robot2GripControl;
   "ST10Cylinder".Cy[15].In.Error := #AlwaysON AND NOT #AlwaysON;
END_REGION

REGION Network 7: CY16 interface F-ROOBT2Gripper2Cylinder
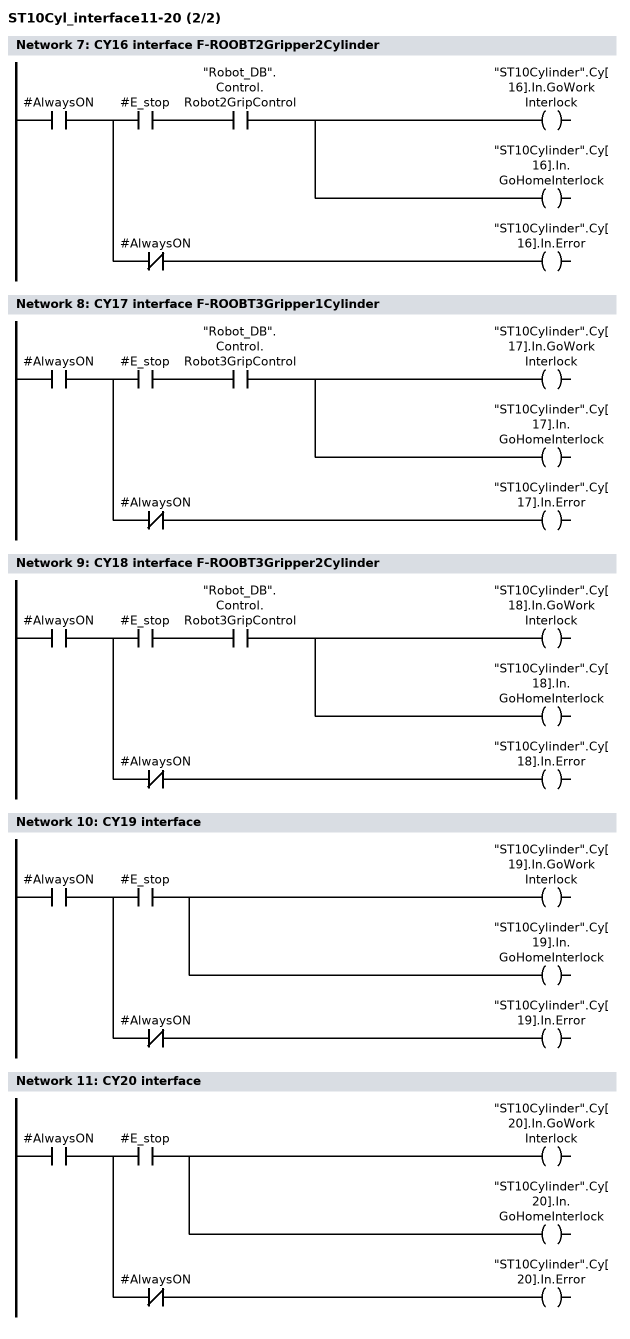
   RUNG wire#powerrail
      Contact( #AlwaysON )
      wire#w1
      Contact( #E_stop )
      Contact( "Robot_DB".Control.Robot2GripControl )
      wire#w2
      Coil( "ST10Cylinder".Cy[16].In.GoWorkInterlock )
   END_RUNG
   RUNG wire#w2
      Coil( "ST10Cylinder".Cy[16].In.GoHomeInterlock )
   END_RUNG
   RUNG wire#w1
      I_Contact( #AlwaysON )
      Coil( "ST10Cylinder".Cy[16].In.Error )
   END_RUNG
   // the same network as SCL:
   "ST10Cylinder".Cy[16].In.GoWorkInterlock := #AlwaysON AND #E_stop AND "Robot_DB".Control.Robot2GripControl;
   "ST10Cylinder".Cy[16].In.GoHomeInterlock := #AlwaysON AND #E_stop AND "Robot_DB".Control.Robot2GripControl;
   "ST10Cylinder".Cy[16].In.Error := #AlwaysON AND NOT #AlwaysON;
END_REGION

REGION Network 8: CY17 interface F-ROOBT3Gripper1Cylinder
   RUNG wire#powerrail
      Contact( #AlwaysON )
      wire#w1
      Contact( #E_stop )
      Contact( "Robot_DB".Control.Robot3GripControl )
      wire#w2
      Coil( "ST10Cylinder".Cy[17].In.GoWorkInterlock )
   END_RUNG
   RUNG wire#w2
      Coil( "ST10Cylinder".Cy[17].In.GoHomeInterlock )
   END_RUNG
   RUNG wire#w1
      I_Contact( #AlwaysON )
      Coil( "ST10Cylinder".Cy[17].In.Error )
   END_RUNG
   // the same network as SCL:
   "ST10Cylinder".Cy[17].In.GoWorkInterlock := #AlwaysON AND #E_stop AND "Robot_DB".Control.Robot3GripControl;
   "ST10Cylinder".Cy[17].In.GoHomeInterlock := #AlwaysON AND #E_stop AND "Robot_DB".Control.Robot3GripControl;
   "ST10Cylinder".Cy[17].In.Error := #AlwaysON AND NOT #AlwaysON;
END_REGION

REGION Network 9: CY18 interface F-ROOBT3Gripper2Cylinder
   RUNG wire#powerrail
      Contact( #AlwaysON )
      wire#w1
      Contact( #E_stop )
      Contact( "Robot_DB".Control.Robot3GripControl )
      wire#w2
      Coil( "ST10Cylinder".Cy[18].In.GoWorkInterlock )
   END_RUNG
   RUNG wire#w2
      Coil( "ST10Cylinder".Cy[18].In.GoHomeInterlock )
   END_RUNG
   RUNG wire#w1
      I_Contact( #AlwaysON )
      Coil( "ST10Cylinder".Cy[18].In.Error )
   END_RUNG
   // the same network as SCL:
   "ST10Cylinder".Cy[18].In.GoWorkInterlock := #AlwaysON AND #E_stop AND "Robot_DB".Control.Robot3GripControl;
   "ST10Cylinder".Cy[18].In.GoHomeInterlock := #AlwaysON AND #E_stop AND "Robot_DB".Control.Robot3GripControl;
   "ST10Cylinder".Cy[18].In.Error := #AlwaysON AND NOT #AlwaysON;
END_REGION

REGION Network 10: CY19 interface
   RUNG wire#powerrail
      Contact( #AlwaysON )
      wire#w1
      Contact( #E_stop )
      wire#w2
      Coil( "ST10Cylinder".Cy[19].In.GoWorkInterlock )
   END_RUNG
   RUNG wire#w2
      Coil( "ST10Cylinder".Cy[19].In.GoHomeInterlock )
   END_RUNG
   RUNG wire#w1
      I_Contact( #AlwaysON )
      Coil( "ST10Cylinder".Cy[19].In.Error )
   END_RUNG
   // the same network as SCL:
   "ST10Cylinder".Cy[19].In.GoWorkInterlock := #AlwaysON AND #E_stop;
   "ST10Cylinder".Cy[19].In.GoHomeInterlock := #AlwaysON AND #E_stop;
   "ST10Cylinder".Cy[19].In.Error := #AlwaysON AND NOT #AlwaysON;
END_REGION

REGION Network 11: CY20 interface
   RUNG wire#powerrail
      Contact( #AlwaysON )
      wire#w1
      Contact( #E_stop )
      wire#w2
      Coil( "ST10Cylinder".Cy[20].In.GoWorkInterlock )
   END_RUNG
   RUNG wire#w2
      Coil( "ST10Cylinder".Cy[20].In.GoHomeInterlock )
   END_RUNG
   RUNG wire#w1
      I_Contact( #AlwaysON )
      Coil( "ST10Cylinder".Cy[20].In.Error )
   END_RUNG
   // the same network as SCL:
   "ST10Cylinder".Cy[20].In.GoWorkInterlock := #AlwaysON AND #E_stop;
   "ST10Cylinder".Cy[20].In.GoHomeInterlock := #AlwaysON AND #E_stop;
   "ST10Cylinder".Cy[20].In.Error := #AlwaysON AND NOT #AlwaysON;
END_REGION
END_FUNCTION

FUNCTION "ST10Cyl_interface31-40" : Void   // FC1023, LAD
{ S7_Optimized_Access := 'FALSE' }
// stored: AutoNumber false, SetENOAutomatically false
   VAR_INPUT
      AlwaysON : Bool;
      E_stop : Bool;
   END_VAR
   VAR_TEMP
      tTest : Bool;
   END_VAR
BEGIN

REGION Network 1 (SCL): Cylinder 31-40 IO Interface (SCL)

   //Cylinder31 IO  J-magnetLiftingLiftingCylinder
   //Input
   "ST10Cylinder".Cy[31].In.WorkPositionSensor := "iJ-magnetLiftingLiftingCylinderInWP";
   "ST10Cylinder".Cy[31].In.HomePositionSensor := "iJ-magnetLiftingLiftingCylinderInHP";
   //Output
   "oJ-magnetLiftingLiftingCylinderToWP" := "ST10Cylinder".Cy[31].Out.GoWorkPosition;
   "oJ-magnetLiftingLiftingCylinderToHP" := "ST10Cylinder".Cy[31].Out.GoHomePosition;

   //Cylinder32 IO  J-magnetLiftingPalletLocationCylinder
   //Input
   "ST10Cylinder".Cy[32].In.WorkPositionSensor := "iJ-magnetLiftingPalletLocationCylinderInWP";
   "ST10Cylinder".Cy[32].In.HomePositionSensor := "iJ-magnetLiftingPalletLocationCylinderInHP";
   //Output
   "oJ-magnetLiftingPalletLocationCylinderToWP" := "ST10Cylinder".Cy[32].Out.GoWorkPosition;
   "oJ-magnetLiftingPalletLocationCylinderToHP" := "ST10Cylinder".Cy[32].Out.GoHomePosition;

   //Cylinder33 IO  J-magnetLoadingStopperCylinder1
   //Input
   "ST10Cylinder".Cy[33].In.WorkPositionSensor := "oJ-magnetLoadingStopperCylinder1_ToWP";
   "ST10Cylinder".Cy[33].In.HomePositionSensor := "oJ-magnetLoadingStopperCylinder1_ToHP";
   //Output
   "oJ-magnetLoadingStopperCylinder1_ToWP" := "ST10Cylinder".Cy[33].Out.GoWorkPosition;
   "oJ-magnetLoadingStopperCylinder1_ToHP" := "ST10Cylinder".Cy[33].Out.GoHomePosition;

   //Cylinder34 IO  J-magnetLoadingStopperCylinder2
   //Input
   "ST10Cylinder".Cy[34].In.WorkPositionSensor := "oJ-magnetLoadingStopperCylinder2_ToWP";
   "ST10Cylinder".Cy[34].In.HomePositionSensor := "oJ-magnetLoadingStopperCylinder2_ToHP";
   //Output
   "oJ-magnetLoadingStopperCylinder2_ToWP" := "ST10Cylinder".Cy[34].Out.GoWorkPosition;
   "oJ-magnetLoadingStopperCylinder2_ToHP" := "ST10Cylinder".Cy[34].Out.GoHomePosition;

   //Cylinder35 IO  J-magnetLoadingStopperCylinder3
   //Input
   "ST10Cylinder".Cy[35].In.WorkPositionSensor := "oJ-magnetLoadingStopperCylinder3_ToWP";
   "ST10Cylinder".Cy[35].In.HomePositionSensor := "oJ-magnetLoadingStopperCylinder3_ToHP";
   //Output
   "oJ-magnetLoadingStopperCylinder3_ToWP" := "ST10Cylinder".Cy[35].Out.GoWorkPosition;
   "oJ-magnetLoadingStopperCylinder3_ToHP" := "ST10Cylinder".Cy[35].Out.GoHomePosition;

   //Cylinder36 J-magnetLoadingStopperCylinder4
   //Input
   "ST10Cylinder".Cy[36].In.WorkPositionSensor := "oJ-magnetLoadingStopperCylinder4_ToWP";
   "ST10Cylinder".Cy[36].In.HomePositionSensor := "oJ-magnetLoadingStopperCylinder4_ToHP";
   //Output
   "oJ-magnetLoadingStopperCylinder4_ToWP" := "ST10Cylinder".Cy[36].Out.GoWorkPosition;
   "oJ-magnetLoadingStopperCylinder4_ToHP" := "ST10Cylinder".Cy[36].Out.GoHomePosition;

   //Cylinder37 J-magnetTakeStopperCylinder1
   //Input
   "ST10Cylinder".Cy[37].In.WorkPositionSensor := "oJ-magnetTakeStopperCylinder1_ToWP";
   "ST10Cylinder".Cy[37].In.HomePositionSensor := "oJ-magnetTakeStopperCylinder1_ToHP";
   //Output
   "oJ-magnetTakeStopperCylinder1_ToWP" := "ST10Cylinder".Cy[37].Out.GoWorkPosition;
   "oJ-magnetTakeStopperCylinder1_ToHP" := "ST10Cylinder".Cy[37].Out.GoHomePosition;

   //Cylinder38 J-magnetTakeStopperCylinder2
   //Input
   "ST10Cylinder".Cy[38].In.WorkPositionSensor := "oJ-magnetTakeStopperCylinder2_ToWP";
   "ST10Cylinder".Cy[38].In.HomePositionSensor := "oJ-magnetTakeStopperCylinder2_ToHP";
   //Output
   "oJ-magnetTakeStopperCylinder2_ToWP" := "ST10Cylinder".Cy[38].Out.GoWorkPosition;
   "oJ-magnetTakeStopperCylinder2_ToHP" := "ST10Cylinder".Cy[38].Out.GoHomePosition;

   //Cylinder39 J-magnetTakeStopperCylinder3
   //Input
   "ST10Cylinder".Cy[39].In.WorkPositionSensor := "oJ-magnetTakeStopperCylinder3_ToWP";
   "ST10Cylinder".Cy[39].In.HomePositionSensor := "oJ-magnetTakeStopperCylinder3_ToHP";
   //Output
   "oJ-magnetTakeStopperCylinder3_ToWP" := "ST10Cylinder".Cy[39].Out.GoWorkPosition;
   "oJ-magnetTakeStopperCylinder3_ToHP" := "ST10Cylinder".Cy[39].Out.GoHomePosition;

   (*
   //Cylinder40 J-magnetLoadingStopperCylinder4_2
   // //Input
   "ST10Cylinder".Cy[40].In.WorkPositionSensor := "oJ-magnetLoadingStopperCylinder4_2";
   "ST10Cylinder".Cy[40].In.HomePositionSensor := NOT "oJ-magnetLoadingStopperCylinder4_2";
   // //Output
   "oJ-magnetLoadingStopperCylinder4_2" := "ST10Cylinder".Cy[40].Out.GoWorkPosition;
   "Feeding washer  lift Cylinder ToHP" := "ST10Cylinder".Cy[40].Out.GoHomePosition;
   *)
END_REGION

REGION Network 2: CY31 interface J-magnetLiftingLiftingCylinder
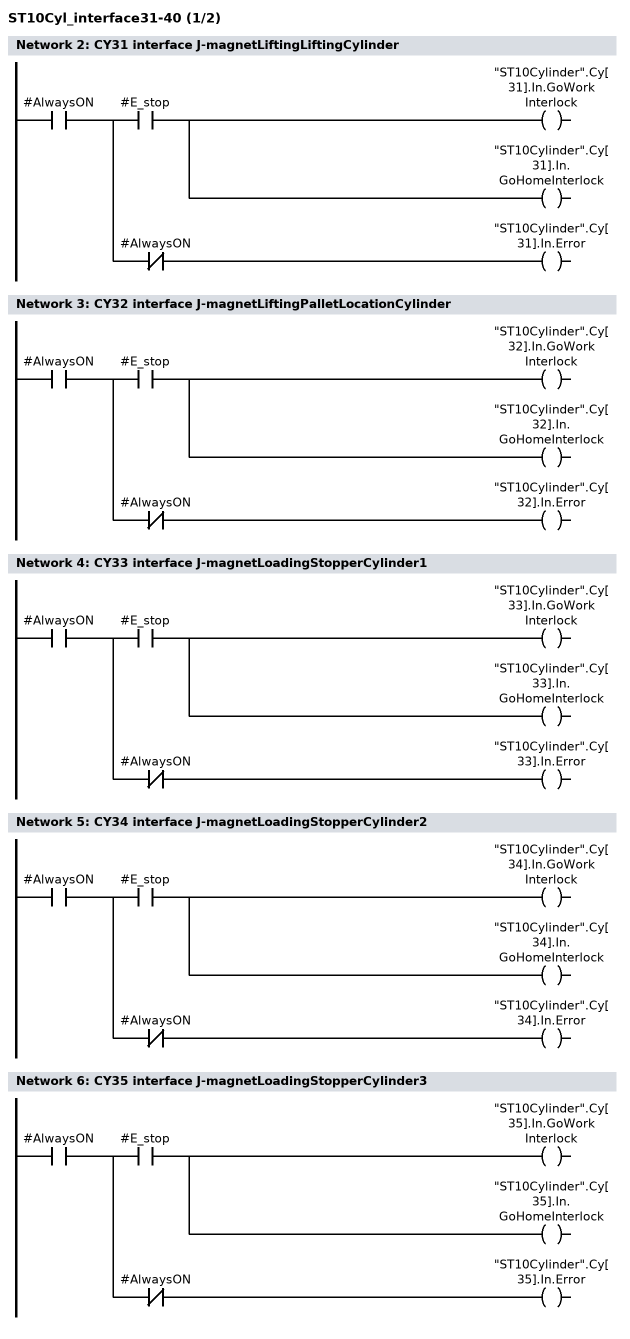
   RUNG wire#powerrail
      Contact( #AlwaysON )
      wire#w1
      Contact( #E_stop )
      wire#w2
      Coil( "ST10Cylinder".Cy[31].In.GoWorkInterlock )
   END_RUNG
   RUNG wire#w2
      Coil( "ST10Cylinder".Cy[31].In.GoHomeInterlock )
   END_RUNG
   RUNG wire#w1
      I_Contact( #AlwaysON )
      Coil( "ST10Cylinder".Cy[31].In.Error )
   END_RUNG
   // the same network as SCL:
   "ST10Cylinder".Cy[31].In.GoWorkInterlock := #AlwaysON AND #E_stop;
   "ST10Cylinder".Cy[31].In.GoHomeInterlock := #AlwaysON AND #E_stop;
   "ST10Cylinder".Cy[31].In.Error := #AlwaysON AND NOT #AlwaysON;
END_REGION

REGION Network 3: CY32 interface J-magnetLiftingPalletLocationCylinder
   RUNG wire#powerrail
      Contact( #AlwaysON )
      wire#w1
      Contact( #E_stop )
      wire#w2
      Coil( "ST10Cylinder".Cy[32].In.GoWorkInterlock )
   END_RUNG
   RUNG wire#w2
      Coil( "ST10Cylinder".Cy[32].In.GoHomeInterlock )
   END_RUNG
   RUNG wire#w1
      I_Contact( #AlwaysON )
      Coil( "ST10Cylinder".Cy[32].In.Error )
   END_RUNG
   // the same network as SCL:
   "ST10Cylinder".Cy[32].In.GoWorkInterlock := #AlwaysON AND #E_stop;
   "ST10Cylinder".Cy[32].In.GoHomeInterlock := #AlwaysON AND #E_stop;
   "ST10Cylinder".Cy[32].In.Error := #AlwaysON AND NOT #AlwaysON;
END_REGION

REGION Network 4: CY33 interface J-magnetLoadingStopperCylinder1
   RUNG wire#powerrail
      Contact( #AlwaysON )
      wire#w1
      Contact( #E_stop )
      wire#w2
      Coil( "ST10Cylinder".Cy[33].In.GoWorkInterlock )
   END_RUNG
   RUNG wire#w2
      Coil( "ST10Cylinder".Cy[33].In.GoHomeInterlock )
   END_RUNG
   RUNG wire#w1
      I_Contact( #AlwaysON )
      Coil( "ST10Cylinder".Cy[33].In.Error )
   END_RUNG
   // the same network as SCL:
   "ST10Cylinder".Cy[33].In.GoWorkInterlock := #AlwaysON AND #E_stop;
   "ST10Cylinder".Cy[33].In.GoHomeInterlock := #AlwaysON AND #E_stop;
   "ST10Cylinder".Cy[33].In.Error := #AlwaysON AND NOT #AlwaysON;
END_REGION

REGION Network 5: CY34 interface J-magnetLoadingStopperCylinder2
   RUNG wire#powerrail
      Contact( #AlwaysON )
      wire#w1
      Contact( #E_stop )
      wire#w2
      Coil( "ST10Cylinder".Cy[34].In.GoWorkInterlock )
   END_RUNG
   RUNG wire#w2
      Coil( "ST10Cylinder".Cy[34].In.GoHomeInterlock )
   END_RUNG
   RUNG wire#w1
      I_Contact( #AlwaysON )
      Coil( "ST10Cylinder".Cy[34].In.Error )
   END_RUNG
   // the same network as SCL:
   "ST10Cylinder".Cy[34].In.GoWorkInterlock := #AlwaysON AND #E_stop;
   "ST10Cylinder".Cy[34].In.GoHomeInterlock := #AlwaysON AND #E_stop;
   "ST10Cylinder".Cy[34].In.Error := #AlwaysON AND NOT #AlwaysON;
END_REGION

REGION Network 6: CY35 interface J-magnetLoadingStopperCylinder3
   RUNG wire#powerrail
      Contact( #AlwaysON )
      wire#w1
      Contact( #E_stop )
      wire#w2
      Coil( "ST10Cylinder".Cy[35].In.GoWorkInterlock )
   END_RUNG
   RUNG wire#w2
      Coil( "ST10Cylinder".Cy[35].In.GoHomeInterlock )
   END_RUNG
   RUNG wire#w1
      I_Contact( #AlwaysON )
      Coil( "ST10Cylinder".Cy[35].In.Error )
   END_RUNG
   // the same network as SCL:
   "ST10Cylinder".Cy[35].In.GoWorkInterlock := #AlwaysON AND #E_stop;
   "ST10Cylinder".Cy[35].In.GoHomeInterlock := #AlwaysON AND #E_stop;
   "ST10Cylinder".Cy[35].In.Error := #AlwaysON AND NOT #AlwaysON;
END_REGION

REGION Network 7: CY36 interface J-magnetLoadingStopperCylinder4
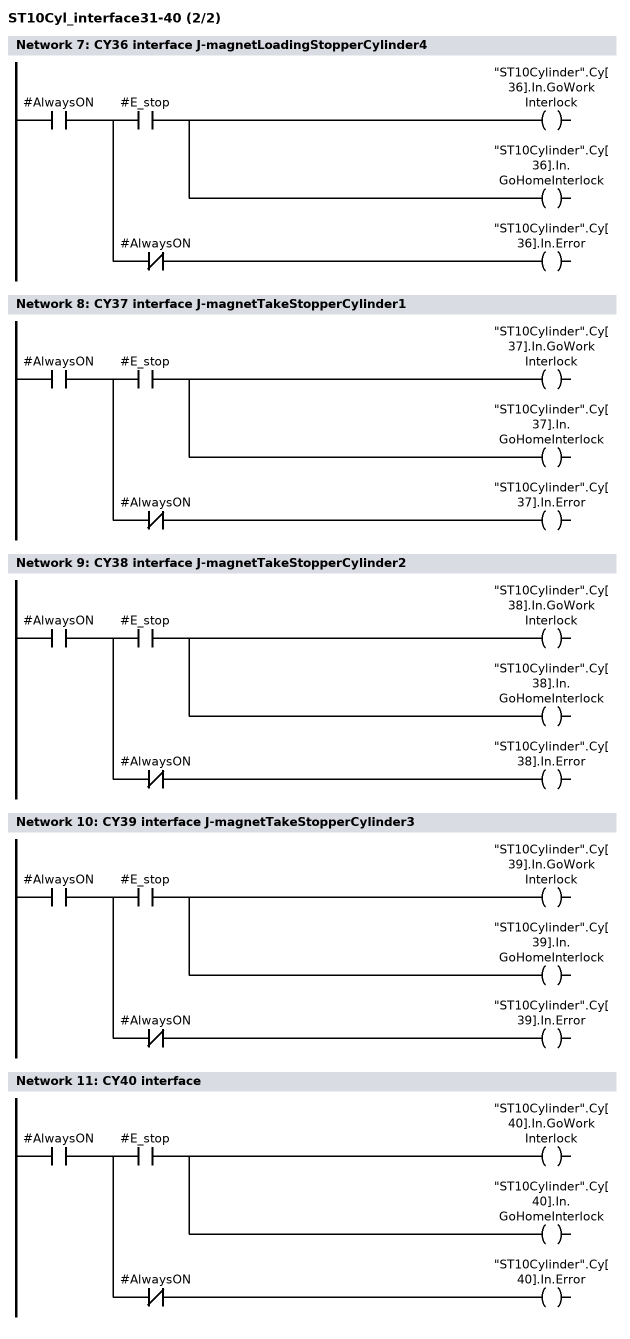
   RUNG wire#powerrail
      Contact( #AlwaysON )
      wire#w1
      Contact( #E_stop )
      wire#w2
      Coil( "ST10Cylinder".Cy[36].In.GoWorkInterlock )
   END_RUNG
   RUNG wire#w2
      Coil( "ST10Cylinder".Cy[36].In.GoHomeInterlock )
   END_RUNG
   RUNG wire#w1
      I_Contact( #AlwaysON )
      Coil( "ST10Cylinder".Cy[36].In.Error )
   END_RUNG
   // the same network as SCL:
   "ST10Cylinder".Cy[36].In.GoWorkInterlock := #AlwaysON AND #E_stop;
   "ST10Cylinder".Cy[36].In.GoHomeInterlock := #AlwaysON AND #E_stop;
   "ST10Cylinder".Cy[36].In.Error := #AlwaysON AND NOT #AlwaysON;
END_REGION

REGION Network 8: CY37 interface J-magnetTakeStopperCylinder1
   RUNG wire#powerrail
      Contact( #AlwaysON )
      wire#w1
      Contact( #E_stop )
      wire#w2
      Coil( "ST10Cylinder".Cy[37].In.GoWorkInterlock )
   END_RUNG
   RUNG wire#w2
      Coil( "ST10Cylinder".Cy[37].In.GoHomeInterlock )
   END_RUNG
   RUNG wire#w1
      I_Contact( #AlwaysON )
      Coil( "ST10Cylinder".Cy[37].In.Error )
   END_RUNG
   // the same network as SCL:
   "ST10Cylinder".Cy[37].In.GoWorkInterlock := #AlwaysON AND #E_stop;
   "ST10Cylinder".Cy[37].In.GoHomeInterlock := #AlwaysON AND #E_stop;
   "ST10Cylinder".Cy[37].In.Error := #AlwaysON AND NOT #AlwaysON;
END_REGION

REGION Network 9: CY38 interface J-magnetTakeStopperCylinder2
   RUNG wire#powerrail
      Contact( #AlwaysON )
      wire#w1
      Contact( #E_stop )
      wire#w2
      Coil( "ST10Cylinder".Cy[38].In.GoWorkInterlock )
   END_RUNG
   RUNG wire#w2
      Coil( "ST10Cylinder".Cy[38].In.GoHomeInterlock )
   END_RUNG
   RUNG wire#w1
      I_Contact( #AlwaysON )
      Coil( "ST10Cylinder".Cy[38].In.Error )
   END_RUNG
   // the same network as SCL:
   "ST10Cylinder".Cy[38].In.GoWorkInterlock := #AlwaysON AND #E_stop;
   "ST10Cylinder".Cy[38].In.GoHomeInterlock := #AlwaysON AND #E_stop;
   "ST10Cylinder".Cy[38].In.Error := #AlwaysON AND NOT #AlwaysON;
END_REGION

REGION Network 10: CY39 interface J-magnetTakeStopperCylinder3
   RUNG wire#powerrail
      Contact( #AlwaysON )
      wire#w1
      Contact( #E_stop )
      wire#w2
      Coil( "ST10Cylinder".Cy[39].In.GoWorkInterlock )
   END_RUNG
   RUNG wire#w2
      Coil( "ST10Cylinder".Cy[39].In.GoHomeInterlock )
   END_RUNG
   RUNG wire#w1
      I_Contact( #AlwaysON )
      Coil( "ST10Cylinder".Cy[39].In.Error )
   END_RUNG
   // the same network as SCL:
   "ST10Cylinder".Cy[39].In.GoWorkInterlock := #AlwaysON AND #E_stop;
   "ST10Cylinder".Cy[39].In.GoHomeInterlock := #AlwaysON AND #E_stop;
   "ST10Cylinder".Cy[39].In.Error := #AlwaysON AND NOT #AlwaysON;
END_REGION

REGION Network 11: CY40 interface
   RUNG wire#powerrail
      Contact( #AlwaysON )
      wire#w1
      Contact( #E_stop )
      wire#w2
      Coil( "ST10Cylinder".Cy[40].In.GoWorkInterlock )
   END_RUNG
   RUNG wire#w2
      Coil( "ST10Cylinder".Cy[40].In.GoHomeInterlock )
   END_RUNG
   RUNG wire#w1
      I_Contact( #AlwaysON )
      Coil( "ST10Cylinder".Cy[40].In.Error )
   END_RUNG
   // the same network as SCL:
   "ST10Cylinder".Cy[40].In.GoWorkInterlock := #AlwaysON AND #E_stop;
   "ST10Cylinder".Cy[40].In.GoHomeInterlock := #AlwaysON AND #E_stop;
   "ST10Cylinder".Cy[40].In.Error := #AlwaysON AND NOT #AlwaysON;
END_REGION
END_FUNCTION

FUNCTION "ST10Cyl_interface81-90" : Void   // FC1028, LAD
{ S7_Optimized_Access := 'FALSE' }
// stored: AutoNumber false, SetENOAutomatically false
   VAR_INPUT
      AlwaysON : Bool;
      E_stop : Bool;
   END_VAR
   VAR_TEMP
      tTest : Bool;
   END_VAR
BEGIN

REGION Network 1 (SCL): Cylinder 81-90 IO Interface (SCL)
   (*
   //Cylinder81 IO  L-UnloadingTransCylinder
   //Input
   "ST10Cylinder".Cy[81].In.WorkPositionSensor := "iL-UnloadingTransCylinderInWP";
   "ST10Cylinder".Cy[81].In.HomePositionSensor := "iL-UnloadingTransCylinderInHP";
   //Output
   "oL-UnloadingTransCylinderToWP" := "ST10Cylinder".Cy[81].Out.GoWorkPosition;
   "oL-UnloadingTransCylinderToHP" := "ST10Cylinder".Cy[81].Out.GoHomePosition;

   //Cylinder82 IO  L-UnloadingTransPalletLocationCylinder
   //Input
   "ST10Cylinder".Cy[82].In.WorkPositionSensor := "iL-UnloadingTransPalletLocationCylinderInWP";
   "ST10Cylinder".Cy[82].In.HomePositionSensor := "iL-UnloadingTransPalletLocationCylinderInHP";
   //Output
   "oL-UnloadingTransPalletLocationCylinderToWP" := "ST10Cylinder".Cy[82].Out.GoWorkPosition;
   "oL-UnloadingTransPalletLocationCylinderToHP" := "ST10Cylinder".Cy[82].Out.GoHomePosition;

   //Cylinder83 IO  L-UnloadingStopperCylinder1_1
   //Input
   "ST10Cylinder".Cy[83].In.WorkPositionSensor := "oL-UnloadingStopperCylinder1_1";
   "ST10Cylinder".Cy[83].In.HomePositionSensor := NOT "oL-UnloadingStopperCylinder1_1";
   //Output
   "oL-UnloadingStopperCylinder1_1" := "ST10Cylinder".Cy[83].Out.GoWorkPosition;
   //"oI-0030TrayLoading8trayStopperCylinderToHP" := "ST10Cylinder".Cy[83].Out.GoHomePosition;

   //Cylinder84 IO  L-UnloadingStopperCylinder1_2
   //Input
   "ST10Cylinder".Cy[84].In.WorkPositionSensor := "oL-UnloadingStopperCylinder1_2";
   "ST10Cylinder".Cy[84].In.HomePositionSensor := NOT "oL-UnloadingStopperCylinder1_2";
   //Output
   "oL-UnloadingStopperCylinder1_2" := "ST10Cylinder".Cy[84].Out.GoWorkPosition;
   //"oI-0080TrayLoadingTaketrayCylinderToHP" := "ST10Cylinder".Cy[84].Out.GoHomePosition;

   //Cylinder85 IO  L-UnloadingStopperCylinder2_1
   //Input
   "ST10Cylinder".Cy[85].In.WorkPositionSensor := "oL-UnloadingStopperCylinder2_1";
   "ST10Cylinder".Cy[85].In.HomePositionSensor := NOT "oL-UnloadingStopperCylinder2_1";
   //Output
   "oL-UnloadingStopperCylinder2_1" := "ST10Cylinder".Cy[85].Out.GoWorkPosition;
   //"oI-0050TrayLoadingTrayCylinderToHP" := "ST10Cylinder".Cy[85].Out.GoHomePosition;

   //Cylinder86  L-UnloadingStopperCylinder2_2
   //Input
   "ST10Cylinder".Cy[86].In.WorkPositionSensor := "oL-UnloadingStopperCylinder2_2";
   "ST10Cylinder".Cy[86].In.HomePositionSensor := NOT "oL-UnloadingStopperCylinder2_2";
   //Output
   "oL-UnloadingStopperCylinder2_2" := "ST10Cylinder".Cy[86].Out.GoWorkPosition;
   //"oI-0080TrayLoadingTraySupportCylinder1ToHP" := "ST10Cylinder".Cy[86].Out.GoHomePosition;

   //Cylinder87 L-UnloadingStopperCylinder3_1
   //Input
   "ST10Cylinder".Cy[87].In.WorkPositionSensor := "oL-UnloadingStopperCylinder3_1";
   "ST10Cylinder".Cy[87].In.HomePositionSensor := NOT "oL-UnloadingStopperCylinder3_1";
   //Output
   "oL-UnloadingStopperCylinder3_1" := "ST10Cylinder".Cy[87].Out.GoWorkPosition;
   //"oI-0070TrayLoadingTraySupportCylinder8ToHP" := "ST10Cylinder".Cy[87].Out.GoHomePosition;

   //Cylinder88 L-UnloadingStopperCylinder3_2
   //Input
   "ST10Cylinder".Cy[88].In.WorkPositionSensor := "oL-UnloadingStopperCylinder3_2";
   "ST10Cylinder".Cy[88].In.HomePositionSensor := NOT "oL-UnloadingStopperCylinder3_2";
   //Output
   "oL-UnloadingStopperCylinder3_2" := "ST10Cylinder".Cy[88].Out.GoWorkPosition;
   //"oI-0080TrayLoadingTrayLocationCylinderToHP" := "ST10Cylinder".Cy[88].Out.GoHomePosition;
   //
   *)
   (*
   //Cylinder89 K-reserveLoadingStopperCylinder4_1
   //Input
   "ST10Cylinder".Cy[89].In.WorkPositionSensor := "oK-reserveLoadingStopperCylinder4_1";
   "ST10Cylinder".Cy[89].In.HomePositionSensor := NOT "oK-reserveLoadingStopperCylinder4_1";
   //Output
   "oK-reserveLoadingStopperCylinder4_1" := "ST10Cylinder".Cy[89].Out.GoWorkPosition;
   //"oI-0090TrayLoadingTrayUnloadingLiftingCylinderToHP" := "ST10Cylinder".Cy[89].Out.GoHomePosition;

   //Cylinder70 K-reserveLoadingStopperCylinder4_2
   // //Input
   "ST10Cylinder".Cy[70].In.WorkPositionSensor := "oK-reserveLoadingStopperCylinder4_2";
   "ST10Cylinder".Cy[70].In.HomePositionSensor := NOT "oK-reserveLoadingStopperCylinder4_2";
   // //Output
   "oK-reserveLoadingStopperCylinder4_2" := "ST10Cylinder".Cy[70].Out.GoWorkPosition;
   // "Feeding washer  lift Cylinder ToHP" := "ST10Cylinder".Cy[70].Out.GoHomePosition;

   *)
END_REGION

REGION Network 2: CY81 interface L-UnloadingTransCylinder
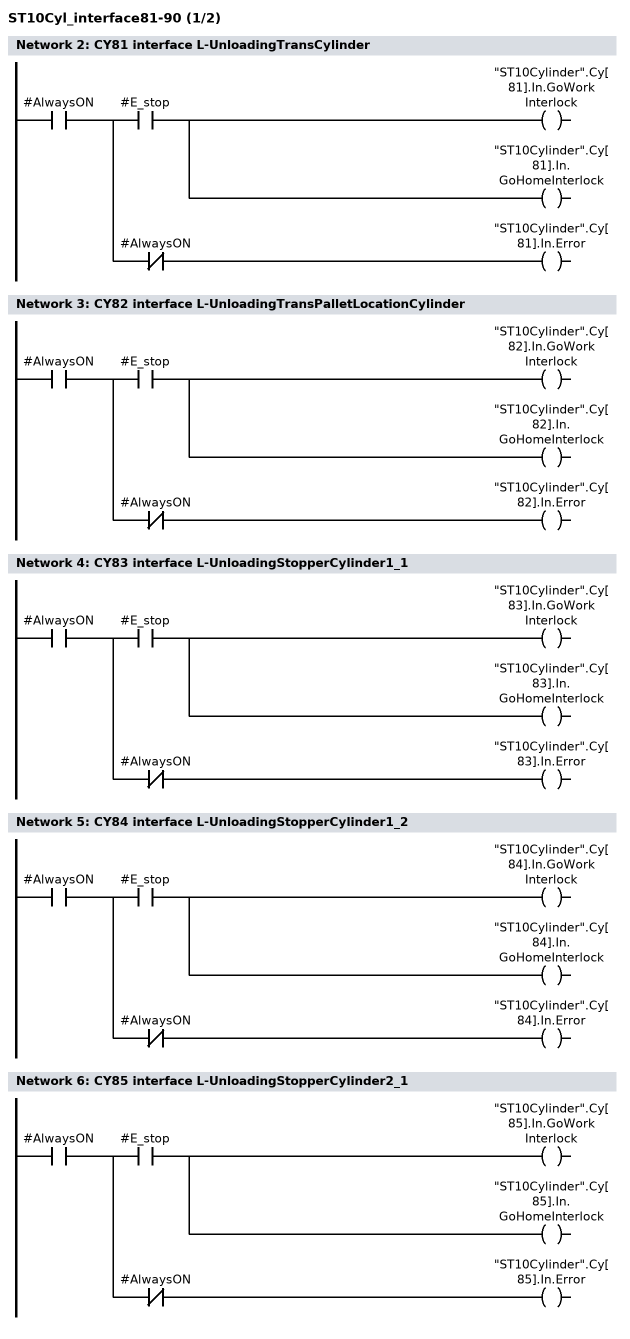
   RUNG wire#powerrail
      Contact( #AlwaysON )
      wire#w1
      Contact( #E_stop )
      wire#w2
      Coil( "ST10Cylinder".Cy[81].In.GoWorkInterlock )
   END_RUNG
   RUNG wire#w2
      Coil( "ST10Cylinder".Cy[81].In.GoHomeInterlock )
   END_RUNG
   RUNG wire#w1
      I_Contact( #AlwaysON )
      Coil( "ST10Cylinder".Cy[81].In.Error )
   END_RUNG
   // the same network as SCL:
   "ST10Cylinder".Cy[81].In.GoWorkInterlock := #AlwaysON AND #E_stop;
   "ST10Cylinder".Cy[81].In.GoHomeInterlock := #AlwaysON AND #E_stop;
   "ST10Cylinder".Cy[81].In.Error := #AlwaysON AND NOT #AlwaysON;
END_REGION

REGION Network 3: CY82 interface L-UnloadingTransPalletLocationCylinder
   RUNG wire#powerrail
      Contact( #AlwaysON )
      wire#w1
      Contact( #E_stop )
      wire#w2
      Coil( "ST10Cylinder".Cy[82].In.GoWorkInterlock )
   END_RUNG
   RUNG wire#w2
      Coil( "ST10Cylinder".Cy[82].In.GoHomeInterlock )
   END_RUNG
   RUNG wire#w1
      I_Contact( #AlwaysON )
      Coil( "ST10Cylinder".Cy[82].In.Error )
   END_RUNG
   // the same network as SCL:
   "ST10Cylinder".Cy[82].In.GoWorkInterlock := #AlwaysON AND #E_stop;
   "ST10Cylinder".Cy[82].In.GoHomeInterlock := #AlwaysON AND #E_stop;
   "ST10Cylinder".Cy[82].In.Error := #AlwaysON AND NOT #AlwaysON;
END_REGION

REGION Network 4: CY83 interface L-UnloadingStopperCylinder1_1
   RUNG wire#powerrail
      Contact( #AlwaysON )
      wire#w1
      Contact( #E_stop )
      wire#w2
      Coil( "ST10Cylinder".Cy[83].In.GoWorkInterlock )
   END_RUNG
   RUNG wire#w2
      Coil( "ST10Cylinder".Cy[83].In.GoHomeInterlock )
   END_RUNG
   RUNG wire#w1
      I_Contact( #AlwaysON )
      Coil( "ST10Cylinder".Cy[83].In.Error )
   END_RUNG
   // the same network as SCL:
   "ST10Cylinder".Cy[83].In.GoWorkInterlock := #AlwaysON AND #E_stop;
   "ST10Cylinder".Cy[83].In.GoHomeInterlock := #AlwaysON AND #E_stop;
   "ST10Cylinder".Cy[83].In.Error := #AlwaysON AND NOT #AlwaysON;
END_REGION

REGION Network 5: CY84 interface L-UnloadingStopperCylinder1_2
   RUNG wire#powerrail
      Contact( #AlwaysON )
      wire#w1
      Contact( #E_stop )
      wire#w2
      Coil( "ST10Cylinder".Cy[84].In.GoWorkInterlock )
   END_RUNG
   RUNG wire#w2
      Coil( "ST10Cylinder".Cy[84].In.GoHomeInterlock )
   END_RUNG
   RUNG wire#w1
      I_Contact( #AlwaysON )
      Coil( "ST10Cylinder".Cy[84].In.Error )
   END_RUNG
   // the same network as SCL:
   "ST10Cylinder".Cy[84].In.GoWorkInterlock := #AlwaysON AND #E_stop;
   "ST10Cylinder".Cy[84].In.GoHomeInterlock := #AlwaysON AND #E_stop;
   "ST10Cylinder".Cy[84].In.Error := #AlwaysON AND NOT #AlwaysON;
END_REGION

REGION Network 6: CY85 interface L-UnloadingStopperCylinder2_1
   RUNG wire#powerrail
      Contact( #AlwaysON )
      wire#w1
      Contact( #E_stop )
      wire#w2
      Coil( "ST10Cylinder".Cy[85].In.GoWorkInterlock )
   END_RUNG
   RUNG wire#w2
      Coil( "ST10Cylinder".Cy[85].In.GoHomeInterlock )
   END_RUNG
   RUNG wire#w1
      I_Contact( #AlwaysON )
      Coil( "ST10Cylinder".Cy[85].In.Error )
   END_RUNG
   // the same network as SCL:
   "ST10Cylinder".Cy[85].In.GoWorkInterlock := #AlwaysON AND #E_stop;
   "ST10Cylinder".Cy[85].In.GoHomeInterlock := #AlwaysON AND #E_stop;
   "ST10Cylinder".Cy[85].In.Error := #AlwaysON AND NOT #AlwaysON;
END_REGION

REGION Network 7: CY86 interface L-UnloadingStopperCylinder2_2
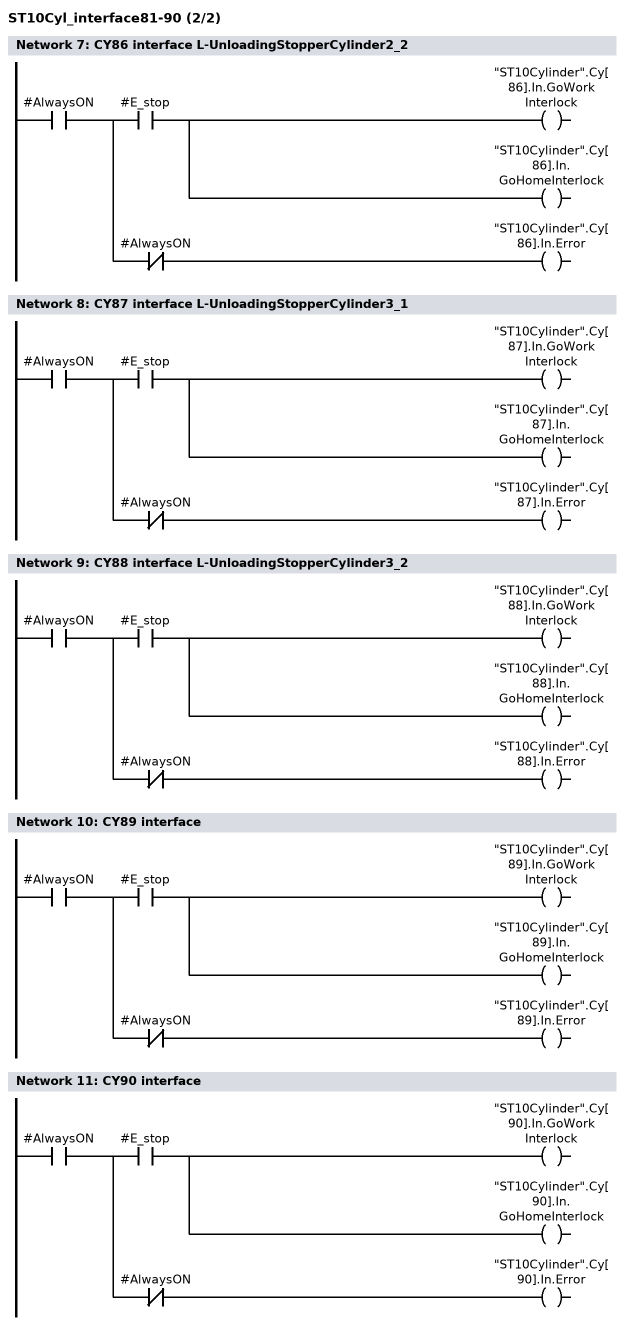
   RUNG wire#powerrail
      Contact( #AlwaysON )
      wire#w1
      Contact( #E_stop )
      wire#w2
      Coil( "ST10Cylinder".Cy[86].In.GoWorkInterlock )
   END_RUNG
   RUNG wire#w2
      Coil( "ST10Cylinder".Cy[86].In.GoHomeInterlock )
   END_RUNG
   RUNG wire#w1
      I_Contact( #AlwaysON )
      Coil( "ST10Cylinder".Cy[86].In.Error )
   END_RUNG
   // the same network as SCL:
   "ST10Cylinder".Cy[86].In.GoWorkInterlock := #AlwaysON AND #E_stop;
   "ST10Cylinder".Cy[86].In.GoHomeInterlock := #AlwaysON AND #E_stop;
   "ST10Cylinder".Cy[86].In.Error := #AlwaysON AND NOT #AlwaysON;
END_REGION

REGION Network 8: CY87 interface L-UnloadingStopperCylinder3_1
   RUNG wire#powerrail
      Contact( #AlwaysON )
      wire#w1
      Contact( #E_stop )
      wire#w2
      Coil( "ST10Cylinder".Cy[87].In.GoWorkInterlock )
   END_RUNG
   RUNG wire#w2
      Coil( "ST10Cylinder".Cy[87].In.GoHomeInterlock )
   END_RUNG
   RUNG wire#w1
      I_Contact( #AlwaysON )
      Coil( "ST10Cylinder".Cy[87].In.Error )
   END_RUNG
   // the same network as SCL:
   "ST10Cylinder".Cy[87].In.GoWorkInterlock := #AlwaysON AND #E_stop;
   "ST10Cylinder".Cy[87].In.GoHomeInterlock := #AlwaysON AND #E_stop;
   "ST10Cylinder".Cy[87].In.Error := #AlwaysON AND NOT #AlwaysON;
END_REGION

REGION Network 9: CY88 interface L-UnloadingStopperCylinder3_2
   RUNG wire#powerrail
      Contact( #AlwaysON )
      wire#w1
      Contact( #E_stop )
      wire#w2
      Coil( "ST10Cylinder".Cy[88].In.GoWorkInterlock )
   END_RUNG
   RUNG wire#w2
      Coil( "ST10Cylinder".Cy[88].In.GoHomeInterlock )
   END_RUNG
   RUNG wire#w1
      I_Contact( #AlwaysON )
      Coil( "ST10Cylinder".Cy[88].In.Error )
   END_RUNG
   // the same network as SCL:
   "ST10Cylinder".Cy[88].In.GoWorkInterlock := #AlwaysON AND #E_stop;
   "ST10Cylinder".Cy[88].In.GoHomeInterlock := #AlwaysON AND #E_stop;
   "ST10Cylinder".Cy[88].In.Error := #AlwaysON AND NOT #AlwaysON;
END_REGION

REGION Network 10: CY89 interface
   RUNG wire#powerrail
      Contact( #AlwaysON )
      wire#w1
      Contact( #E_stop )
      wire#w2
      Coil( "ST10Cylinder".Cy[89].In.GoWorkInterlock )
   END_RUNG
   RUNG wire#w2
      Coil( "ST10Cylinder".Cy[89].In.GoHomeInterlock )
   END_RUNG
   RUNG wire#w1
      I_Contact( #AlwaysON )
      Coil( "ST10Cylinder".Cy[89].In.Error )
   END_RUNG
   // the same network as SCL:
   "ST10Cylinder".Cy[89].In.GoWorkInterlock := #AlwaysON AND #E_stop;
   "ST10Cylinder".Cy[89].In.GoHomeInterlock := #AlwaysON AND #E_stop;
   "ST10Cylinder".Cy[89].In.Error := #AlwaysON AND NOT #AlwaysON;
END_REGION

REGION Network 11: CY90 interface
   RUNG wire#powerrail
      Contact( #AlwaysON )
      wire#w1
      Contact( #E_stop )
      wire#w2
      Coil( "ST10Cylinder".Cy[90].In.GoWorkInterlock )
   END_RUNG
   RUNG wire#w2
      Coil( "ST10Cylinder".Cy[90].In.GoHomeInterlock )
   END_RUNG
   RUNG wire#w1
      I_Contact( #AlwaysON )
      Coil( "ST10Cylinder".Cy[90].In.Error )
   END_RUNG
   // the same network as SCL:
   "ST10Cylinder".Cy[90].In.GoWorkInterlock := #AlwaysON AND #E_stop;
   "ST10Cylinder".Cy[90].In.GoHomeInterlock := #AlwaysON AND #E_stop;
   "ST10Cylinder".Cy[90].In.Error := #AlwaysON AND NOT #AlwaysON;
END_REGION
END_FUNCTION

FUNCTION "ST10_Device" : Void   // FC1010, LAD
{ S7_Optimized_Access := 'TRUE' }
// stored: AutoNumber false, SetENOAutomatically false
   VAR_INPUT
      iSysMode : "RCS_SysComInterface_V1";
   END_VAR
BEGIN

NETWORK
TITLE = SafetyGate

      CALL  "ST10_SafetyGate"
      ( iSysMode := #iSysMode
      );


NETWORK
TITLE = PartData

      CALL  "ST10_PartData"
      ( iSysMode := #iSysMode
      );


NETWORK
TITLE = Analog

      CALL  "ST10_Analog"
      ( iSysMode := #iSysMode
      );


REGION Network 4: SR Scan
END_REGION

REGION Network 7: CuringOven
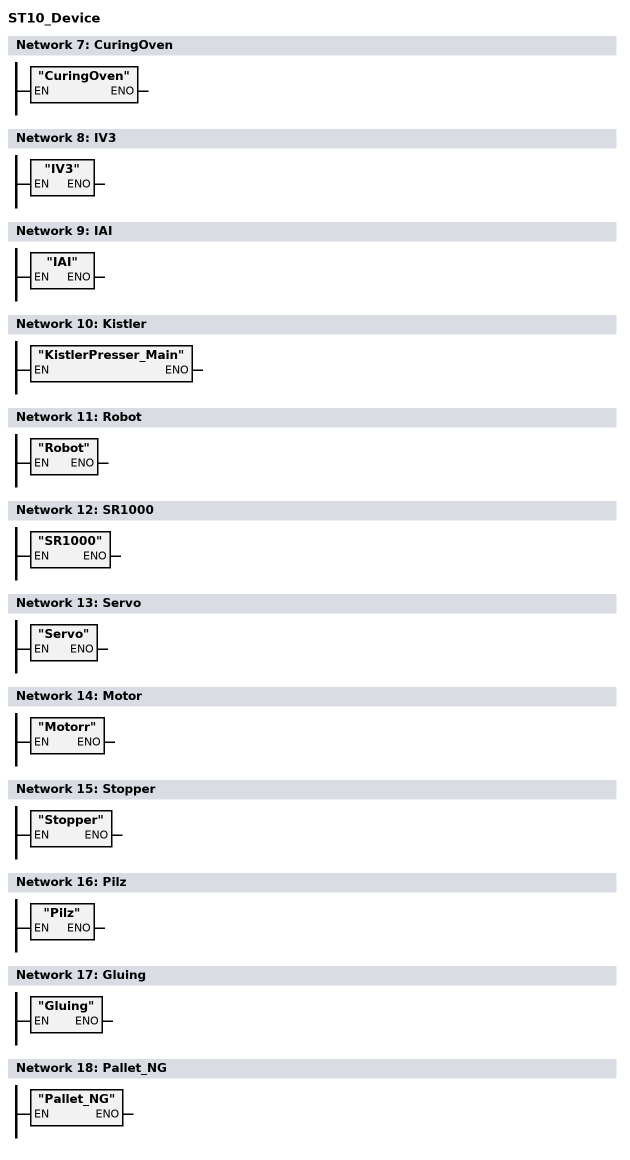
   RUNG wire#powerrail
      "CuringOven"()
   END_RUNG
   // the same network as SCL:
   "CuringOven"();
END_REGION

REGION Network 8: IV3
   RUNG wire#powerrail
      "IV3"()
   END_RUNG
   // the same network as SCL:
   "IV3"();
END_REGION

REGION Network 9: IAI
   RUNG wire#powerrail
      "IAI"()
   END_RUNG
   // the same network as SCL:
   "IAI"();
END_REGION

REGION Network 10: Kistler
   RUNG wire#powerrail
      "KistlerPresser_Main"()
   END_RUNG
   // the same network as SCL:
   "KistlerPresser_Main"();
END_REGION

REGION Network 11: Robot
   RUNG wire#powerrail
      "Robot"()
   END_RUNG
   // the same network as SCL:
   "Robot"();
END_REGION

REGION Network 12: SR1000
   RUNG wire#powerrail
      "SR1000"()
   END_RUNG
   // the same network as SCL:
   "SR1000"();
END_REGION

REGION Network 13: Servo
   RUNG wire#powerrail
      "Servo"()
   END_RUNG
   // the same network as SCL:
   "Servo"();
END_REGION

REGION Network 14: Motor
   RUNG wire#powerrail
      "Motorr"()
   END_RUNG
   // the same network as SCL:
   "Motorr"();
END_REGION

REGION Network 15: Stopper
   RUNG wire#powerrail
      "Stopper"()
   END_RUNG
   // the same network as SCL:
   "Stopper"();
END_REGION

REGION Network 16: Pilz
   RUNG wire#powerrail
      "Pilz"()
   END_RUNG
   // the same network as SCL:
   "Pilz"();
END_REGION

REGION Network 17: Gluing
   RUNG wire#powerrail
      "Gluing"()
   END_RUNG
   // the same network as SCL:
   "Gluing"();
END_REGION

REGION Network 18: Pallet_NG
   RUNG wire#powerrail
      "Pallet_NG"()
   END_RUNG
   // the same network as SCL:
   "Pallet_NG"();
END_REGION
END_FUNCTION

FUNCTION "ST10_Analog" : Void
{ S7_Optimized_Access := 'TRUE' }
VERSION : 0.1
   VAR_INPUT 
      iSysMode : "RCS_SysComInterface_V1";
   END_VAR

   VAR_TEMP 
      idex : Int;
   END_VAR


BEGIN
	
	
	REGION 氮气压模拟量
	    //定义编号
	    #idex := 1;
	    //功能块调用
	
	 END_REGION
	 
	 
	 
	
	 
	 
END_FUNCTION

FUNCTION "SR1000" : Void   // FC1800, LAD
{ S7_Optimized_Access := 'TRUE' }
// stored: AutoNumber false, SetENOAutomatically false
BEGIN

REGION Network 1: 801A1
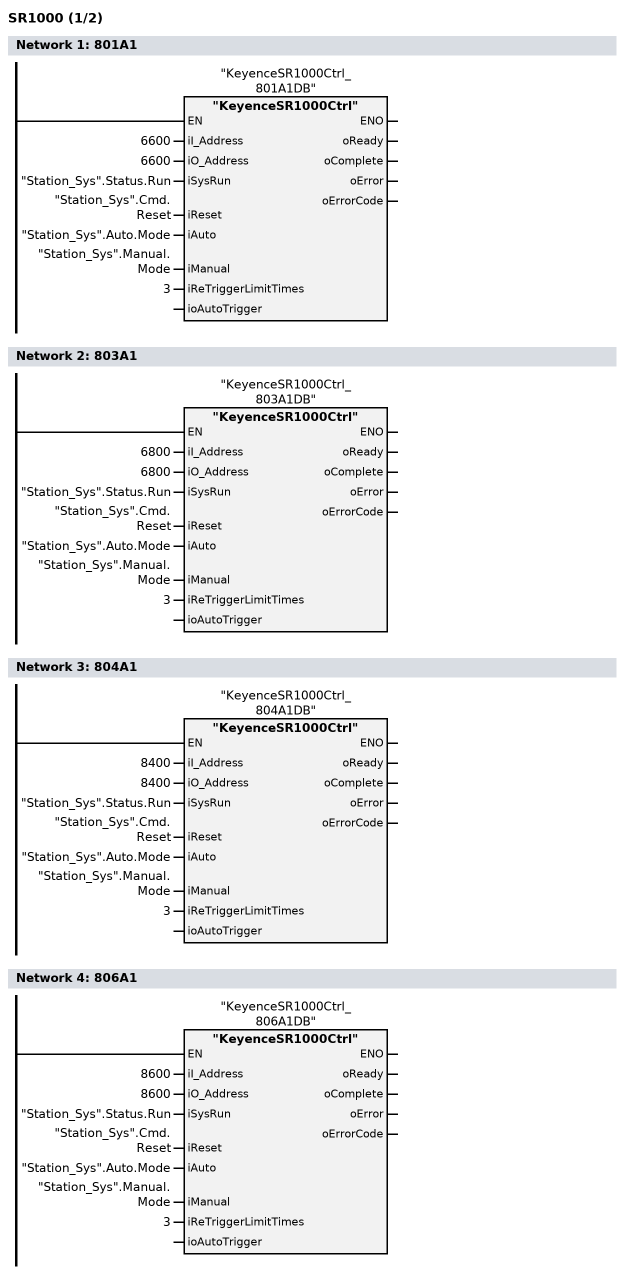
   RUNG wire#powerrail
      "KeyenceSR1000Ctrl_801A1DB"(iI_Address := 6600, iO_Address := 6600, iSysRun := "Station_Sys".Status.Run, iReset := "Station_Sys".Cmd.Reset, iAuto := "Station_Sys".Auto.Mode, iManual := "Station_Sys".Manual.Mode, iReTriggerLimitTimes := 3, ioAutoTrigger :=, oReady =>, oComplete =>, oError =>, oErrorCode =>)
   END_RUNG
   // the same network as SCL:
   "KeyenceSR1000Ctrl_801A1DB"(iI_Address := 6600,   // "KeyenceSR1000Ctrl"
                           iO_Address := 6600,
                           iSysRun := "Station_Sys".Status.Run,
                           iReset := "Station_Sys".Cmd.Reset,
                           iAuto := "Station_Sys".Auto.Mode,
                           iManual := "Station_Sys".Manual.Mode,
                           iReTriggerLimitTimes := 3);
END_REGION

REGION Network 2: 803A1
   RUNG wire#powerrail
      "KeyenceSR1000Ctrl_803A1DB"(iI_Address := 6800, iO_Address := 6800, iSysRun := "Station_Sys".Status.Run, iReset := "Station_Sys".Cmd.Reset, iAuto := "Station_Sys".Auto.Mode, iManual := "Station_Sys".Manual.Mode, iReTriggerLimitTimes := 3, ioAutoTrigger :=, oReady =>, oComplete =>, oError =>, oErrorCode =>)
   END_RUNG
   // the same network as SCL:
   "KeyenceSR1000Ctrl_803A1DB"(iI_Address := 6800,   // "KeyenceSR1000Ctrl"
                           iO_Address := 6800,
                           iSysRun := "Station_Sys".Status.Run,
                           iReset := "Station_Sys".Cmd.Reset,
                           iAuto := "Station_Sys".Auto.Mode,
                           iManual := "Station_Sys".Manual.Mode,
                           iReTriggerLimitTimes := 3);
END_REGION

REGION Network 3: 804A1
   RUNG wire#powerrail
      "KeyenceSR1000Ctrl_804A1DB"(iI_Address := 8400, iO_Address := 8400, iSysRun := "Station_Sys".Status.Run, iReset := "Station_Sys".Cmd.Reset, iAuto := "Station_Sys".Auto.Mode, iManual := "Station_Sys".Manual.Mode, iReTriggerLimitTimes := 3, ioAutoTrigger :=, oReady =>, oComplete =>, oError =>, oErrorCode =>)
   END_RUNG
   // the same network as SCL:
   "KeyenceSR1000Ctrl_804A1DB"(iI_Address := 8400,   // "KeyenceSR1000Ctrl"
                           iO_Address := 8400,
                           iSysRun := "Station_Sys".Status.Run,
                           iReset := "Station_Sys".Cmd.Reset,
                           iAuto := "Station_Sys".Auto.Mode,
                           iManual := "Station_Sys".Manual.Mode,
                           iReTriggerLimitTimes := 3);
END_REGION

REGION Network 4: 806A1
   RUNG wire#powerrail
      "KeyenceSR1000Ctrl_806A1DB"(iI_Address := 8600, iO_Address := 8600, iSysRun := "Station_Sys".Status.Run, iReset := "Station_Sys".Cmd.Reset, iAuto := "Station_Sys".Auto.Mode, iManual := "Station_Sys".Manual.Mode, iReTriggerLimitTimes := 3, ioAutoTrigger :=, oReady =>, oComplete =>, oError =>, oErrorCode =>)
   END_RUNG
   // the same network as SCL:
   "KeyenceSR1000Ctrl_806A1DB"(iI_Address := 8600,   // "KeyenceSR1000Ctrl"
                           iO_Address := 8600,
                           iSysRun := "Station_Sys".Status.Run,
                           iReset := "Station_Sys".Cmd.Reset,
                           iAuto := "Station_Sys".Auto.Mode,
                           iManual := "Station_Sys".Manual.Mode,
                           iReTriggerLimitTimes := 3);
END_REGION

REGION Network 5: 800A1
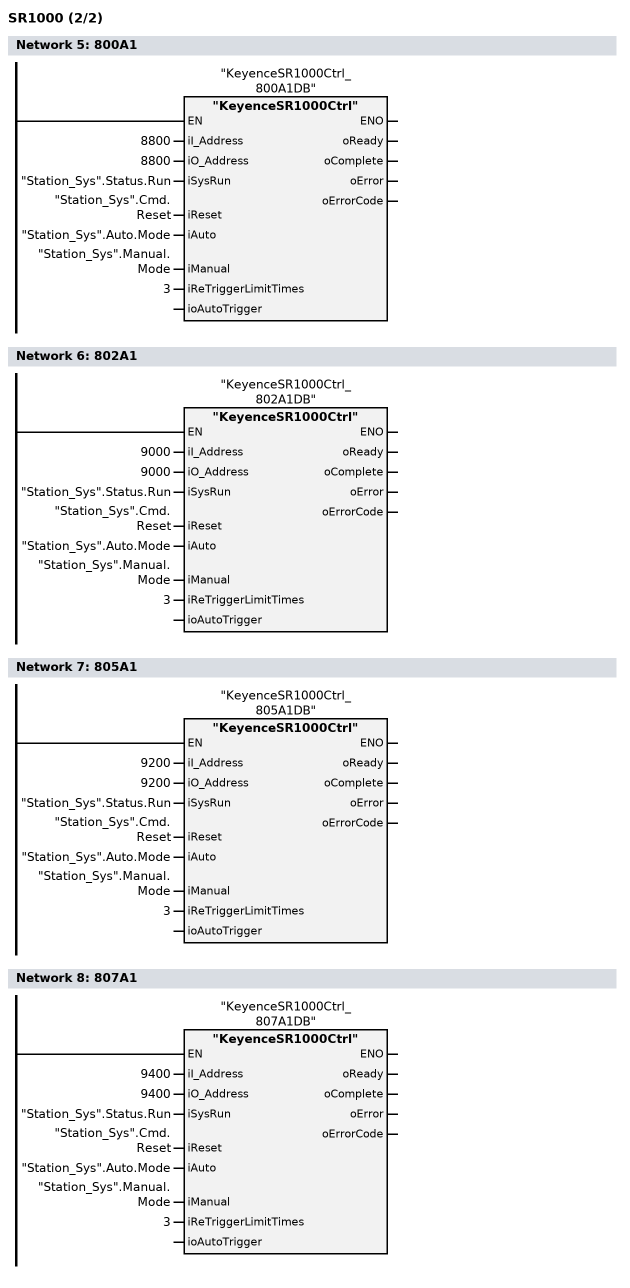
   RUNG wire#powerrail
      "KeyenceSR1000Ctrl_800A1DB"(iI_Address := 8800, iO_Address := 8800, iSysRun := "Station_Sys".Status.Run, iReset := "Station_Sys".Cmd.Reset, iAuto := "Station_Sys".Auto.Mode, iManual := "Station_Sys".Manual.Mode, iReTriggerLimitTimes := 3, ioAutoTrigger :=, oReady =>, oComplete =>, oError =>, oErrorCode =>)
   END_RUNG
   // the same network as SCL:
   "KeyenceSR1000Ctrl_800A1DB"(iI_Address := 8800,   // "KeyenceSR1000Ctrl"
                           iO_Address := 8800,
                           iSysRun := "Station_Sys".Status.Run,
                           iReset := "Station_Sys".Cmd.Reset,
                           iAuto := "Station_Sys".Auto.Mode,
                           iManual := "Station_Sys".Manual.Mode,
                           iReTriggerLimitTimes := 3);
END_REGION

REGION Network 6: 802A1
   RUNG wire#powerrail
      "KeyenceSR1000Ctrl_802A1DB"(iI_Address := 9000, iO_Address := 9000, iSysRun := "Station_Sys".Status.Run, iReset := "Station_Sys".Cmd.Reset, iAuto := "Station_Sys".Auto.Mode, iManual := "Station_Sys".Manual.Mode, iReTriggerLimitTimes := 3, ioAutoTrigger :=, oReady =>, oComplete =>, oError =>, oErrorCode =>)
   END_RUNG
   // the same network as SCL:
   "KeyenceSR1000Ctrl_802A1DB"(iI_Address := 9000,   // "KeyenceSR1000Ctrl"
                           iO_Address := 9000,
                           iSysRun := "Station_Sys".Status.Run,
                           iReset := "Station_Sys".Cmd.Reset,
                           iAuto := "Station_Sys".Auto.Mode,
                           iManual := "Station_Sys".Manual.Mode,
                           iReTriggerLimitTimes := 3);
END_REGION

REGION Network 7: 805A1
   RUNG wire#powerrail
      "KeyenceSR1000Ctrl_805A1DB"(iI_Address := 9200, iO_Address := 9200, iSysRun := "Station_Sys".Status.Run, iReset := "Station_Sys".Cmd.Reset, iAuto := "Station_Sys".Auto.Mode, iManual := "Station_Sys".Manual.Mode, iReTriggerLimitTimes := 3, ioAutoTrigger :=, oReady =>, oComplete =>, oError =>, oErrorCode =>)
   END_RUNG
   // the same network as SCL:
   "KeyenceSR1000Ctrl_805A1DB"(iI_Address := 9200,   // "KeyenceSR1000Ctrl"
                           iO_Address := 9200,
                           iSysRun := "Station_Sys".Status.Run,
                           iReset := "Station_Sys".Cmd.Reset,
                           iAuto := "Station_Sys".Auto.Mode,
                           iManual := "Station_Sys".Manual.Mode,
                           iReTriggerLimitTimes := 3);
END_REGION

REGION Network 8: 807A1
   RUNG wire#powerrail
      "KeyenceSR1000Ctrl_807A1DB"(iI_Address := 9400, iO_Address := 9400, iSysRun := "Station_Sys".Status.Run, iReset := "Station_Sys".Cmd.Reset, iAuto := "Station_Sys".Auto.Mode, iManual := "Station_Sys".Manual.Mode, iReTriggerLimitTimes := 3, ioAutoTrigger :=, oReady =>, oComplete =>, oError =>, oErrorCode =>)
   END_RUNG
   // the same network as SCL:
   "KeyenceSR1000Ctrl_807A1DB"(iI_Address := 9400,   // "KeyenceSR1000Ctrl"
                           iO_Address := 9400,
                           iSysRun := "Station_Sys".Status.Run,
                           iReset := "Station_Sys".Cmd.Reset,
                           iAuto := "Station_Sys".Auto.Mode,
                           iManual := "Station_Sys".Manual.Mode,
                           iReTriggerLimitTimes := 3);
END_REGION
END_FUNCTION

FUNCTION "Servo" : Void   // FC2500, LAD
{ S7_Optimized_Access := 'TRUE' }
// stored: AutoNumber false, SetENOAutomatically false
BEGIN

REGION Network 1
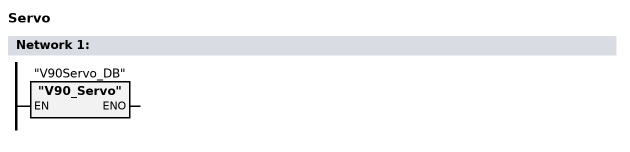
   RUNG wire#powerrail
      "V90Servo_DB"()
   END_RUNG
   // the same network as SCL:
   "V90Servo_DB"();   // "V90_Servo"
END_REGION
END_FUNCTION

FUNCTION "Pallet_NG" : Void   // FC2900, LAD
{ S7_Optimized_Access := 'TRUE' }
// stored: AutoNumber false, SetENOAutomatically false
BEGIN

REGION Network 1
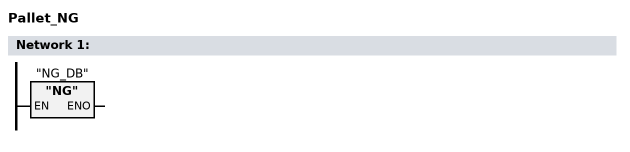
   RUNG wire#powerrail
      "NG_DB"()
   END_RUNG
   // the same network as SCL:
   "NG_DB"();   // "NG"
END_REGION
END_FUNCTION

FUNCTION_BLOCK "NG"   // FB2901, LAD
{ S7_Optimized_Access := 'TRUE' }
// stored: AutoNumber false, MemoryReserve 100, SetENOAutomatically false
   VAR
      NG_L_1 : "NGStatus";
      NG_L_2 { S7_SetPoint := 'True'} : "NGStatus";
      NG_L_3 { S7_SetPoint := 'True'} : "NGStatus";
      NG_UL_1 { S7_SetPoint := 'True'} : "NGStatus";
      NG_UL_2 { S7_SetPoint := 'True'} : "NGStatus";
      NG_UL_3 { S7_SetPoint := 'True'} : "NGStatus";
   END_VAR
   VAR_TEMP   // added for the SCL form of the ladder/FBD networks
      _w1 : Bool;
      _w2 : Bool;
      _w3 : Bool;
      _w4 : Bool;
      _w5 : Bool;
      _w6 : Bool;
      _w7 : Bool;
      _w8 : Bool;
      _w9 : Bool;
      _w10 : Bool;
      _w11 : Bool;
      _w12 : Bool;
      _w13 : Bool;
   END_VAR
BEGIN

REGION Network 1 (SCL): Input
   // NG1
   "PalletNGData".LoadingNGPallet.NG_1_1 := "iE1-UnloadingShaftPressNG_5";
   "PalletNGData".LoadingNGPallet.NG_1_2 := "iE1-UnloadingShaftPressNG_4";
   "PalletNGData".LoadingNGPallet.NG_1_3 := "iE1-UnloadingShaftPressNG_3";
   "PalletNGData".LoadingNGPallet.NG_1_4 := "iE1-UnloadingShaftPressNG_2";
   "PalletNGData".LoadingNGPallet.NG_1_5 := "iE1-UnloadingShaftPressNG_1";

   "PalletNGData".LoadingNGPallet.NG_2_1 := "iE1-UnloadingShaftScanNG_5";
   "PalletNGData".LoadingNGPallet.NG_2_2 := "iE1-UnloadingShaftScanNG_4";
   "PalletNGData".LoadingNGPallet.NG_2_3 := "iE1-UnloadingShaftScanNG_3";
   "PalletNGData".LoadingNGPallet.NG_2_4 := "iE1-UnloadingShaftScanNG_2";
   "PalletNGData".LoadingNGPallet.NG_2_5 := "iE1-UnloadingShaftScanNG_1";

   "PalletNGData".LoadingNGPallet.NG_3_1 := "iE1-UnloadingRingScanNG_5";
   "PalletNGData".LoadingNGPallet.NG_3_2 := "iE1-UnloadingRingScanNG_4";
   "PalletNGData".LoadingNGPallet.NG_3_3 := "iE1-UnloadingRingScanNG_3";
   "PalletNGData".LoadingNGPallet.NG_3_4 := "iE1-UnloadingRingScanNG_2";
   "PalletNGData".LoadingNGPallet.NG_3_5 := "iE1-UnloadingRingScanNG_1";

   // NG2
   "PalletNGData".UnLoadingNGPallet.NG_1_1 := "iE2-UnloadingPressNG_5";
   "PalletNGData".UnLoadingNGPallet.NG_1_2 := "iE2-UnloadingPressNG_4";
   "PalletNGData".UnLoadingNGPallet.NG_1_3 := "iE2-UnloadingPressNG_3";
   "PalletNGData".UnLoadingNGPallet.NG_1_4 := "iE2-UnloadingPressNG_2";
   "PalletNGData".UnLoadingNGPallet.NG_1_5 := "iE2-UnloadingPressNG_1";

   "PalletNGData".UnLoadingNGPallet.NG_2_1 := "iE2-UnloadingMagentScanNG_5";
   "PalletNGData".UnLoadingNGPallet.NG_2_2 := "iE2-UnloadingMagentScanNG_4";
   "PalletNGData".UnLoadingNGPallet.NG_2_3 := "iE2-UnloadingMagentScanNG_3";
   "PalletNGData".UnLoadingNGPallet.NG_2_4 := "iE2-UnloadingMagentScanNG_2";
   "PalletNGData".UnLoadingNGPallet.NG_2_5 := "iE2-UnloadingMagentScanNG_1";

   "PalletNGData".UnLoadingNGPallet.NG_3_1 := "iE2-UnloadingRingScanNG_5";
   "PalletNGData".UnLoadingNGPallet.NG_3_2 := "iE2-UnloadingRingScanNG_4";
   "PalletNGData".UnLoadingNGPallet.NG_3_3 := "iE2-UnloadingRingScanNG_3";
   "PalletNGData".UnLoadingNGPallet.NG_3_4 := "iE2-UnloadingRingScanNG_2";
   "PalletNGData".UnLoadingNGPallet.NG_3_5 := "iE2-UnloadingRingScanNG_1";
END_REGION

REGION Network 2: --------------------------------------- Load -------------------------------------------------------
END_REGION

REGION Network 3: Press
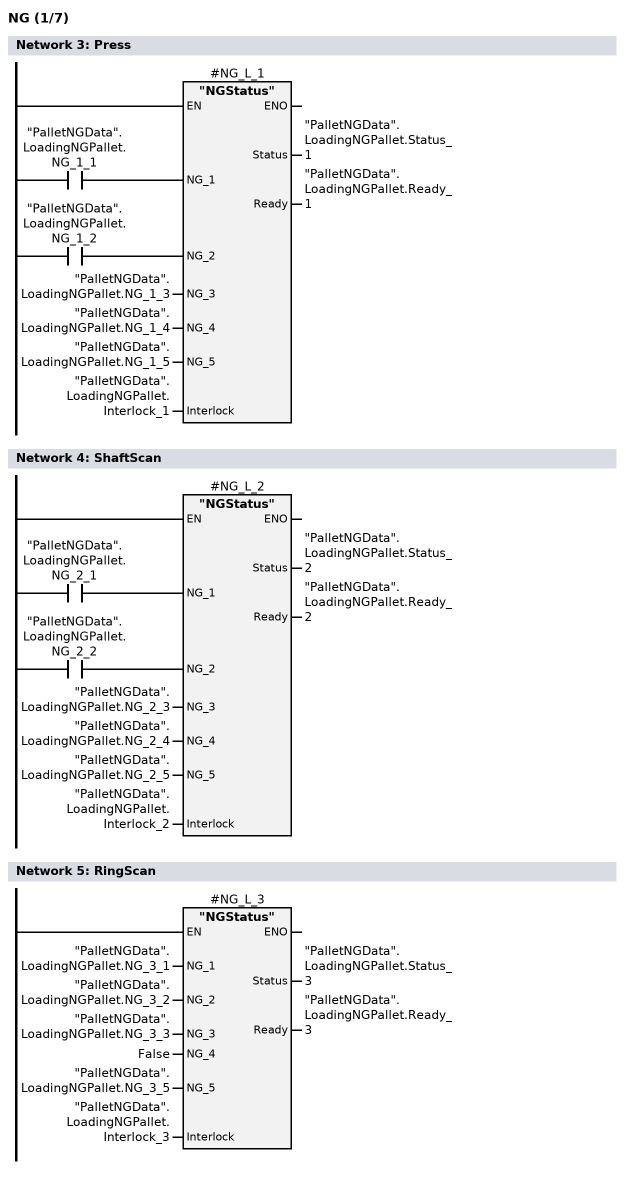
   RUNG wire#powerrail
      #NG_L_1(NG_1 := wire#w1, NG_2 := wire#w2, NG_3 := "PalletNGData".LoadingNGPallet.NG_1_3, NG_4 := "PalletNGData".LoadingNGPallet.NG_1_4, NG_5 := "PalletNGData".LoadingNGPallet.NG_1_5, Interlock := "PalletNGData".LoadingNGPallet.Interlock_1, Status => "PalletNGData".LoadingNGPallet.Status_1, Ready => "PalletNGData".LoadingNGPallet.Ready_1)
   END_RUNG
   RUNG wire#powerrail
      Contact( "PalletNGData".LoadingNGPallet.NG_1_1 )
   END_RUNG wire#w1
   RUNG wire#powerrail
      Contact( "PalletNGData".LoadingNGPallet.NG_1_2 )
   END_RUNG wire#w2
   // the same network as SCL:
   #NG_L_1(NG_1 := "PalletNGData".LoadingNGPallet.NG_1_1,   // "NGStatus"
           NG_2 := "PalletNGData".LoadingNGPallet.NG_1_2,
           NG_3 := "PalletNGData".LoadingNGPallet.NG_1_3,
           NG_4 := "PalletNGData".LoadingNGPallet.NG_1_4,
           NG_5 := "PalletNGData".LoadingNGPallet.NG_1_5,
           Interlock := "PalletNGData".LoadingNGPallet.Interlock_1,
           Status => "PalletNGData".LoadingNGPallet.Status_1,
           Ready => "PalletNGData".LoadingNGPallet.Ready_1);
END_REGION

REGION Network 4: ShaftScan
   RUNG wire#powerrail
      #NG_L_2(NG_1 := wire#w1, NG_2 := wire#w2, NG_3 := "PalletNGData".LoadingNGPallet.NG_2_3, NG_4 := "PalletNGData".LoadingNGPallet.NG_2_4, NG_5 := "PalletNGData".LoadingNGPallet.NG_2_5, Interlock := "PalletNGData".LoadingNGPallet.Interlock_2, Status => "PalletNGData".LoadingNGPallet.Status_2, Ready => "PalletNGData".LoadingNGPallet.Ready_2)
   END_RUNG
   RUNG wire#powerrail
      Contact( "PalletNGData".LoadingNGPallet.NG_2_1 )
   END_RUNG wire#w1
   RUNG wire#powerrail
      Contact( "PalletNGData".LoadingNGPallet.NG_2_2 )
   END_RUNG wire#w2
   // the same network as SCL:
   #NG_L_2(NG_1 := "PalletNGData".LoadingNGPallet.NG_2_1,   // "NGStatus"
           NG_2 := "PalletNGData".LoadingNGPallet.NG_2_2,
           NG_3 := "PalletNGData".LoadingNGPallet.NG_2_3,
           NG_4 := "PalletNGData".LoadingNGPallet.NG_2_4,
           NG_5 := "PalletNGData".LoadingNGPallet.NG_2_5,
           Interlock := "PalletNGData".LoadingNGPallet.Interlock_2,
           Status => "PalletNGData".LoadingNGPallet.Status_2,
           Ready => "PalletNGData".LoadingNGPallet.Ready_2);
END_REGION

REGION Network 5: RingScan
   RUNG wire#powerrail
      #NG_L_3(NG_1 := "PalletNGData".LoadingNGPallet.NG_3_1, NG_2 := "PalletNGData".LoadingNGPallet.NG_3_2, NG_3 := "PalletNGData".LoadingNGPallet.NG_3_3, NG_4 := False, NG_5 := "PalletNGData".LoadingNGPallet.NG_3_5, Interlock := "PalletNGData".LoadingNGPallet.Interlock_3, Status => "PalletNGData".LoadingNGPallet.Status_3, Ready => "PalletNGData".LoadingNGPallet.Ready_3)
   END_RUNG
   // the same network as SCL:
   #NG_L_3(NG_1 := "PalletNGData".LoadingNGPallet.NG_3_1,   // "NGStatus"
           NG_2 := "PalletNGData".LoadingNGPallet.NG_3_2,
           NG_3 := "PalletNGData".LoadingNGPallet.NG_3_3,
           NG_4 := False,
           NG_5 := "PalletNGData".LoadingNGPallet.NG_3_5,
           Interlock := "PalletNGData".LoadingNGPallet.Interlock_3,
           Status => "PalletNGData".LoadingNGPallet.Status_3,
           Ready => "PalletNGData".LoadingNGPallet.Ready_3);
END_REGION

REGION Network 6: InterLock
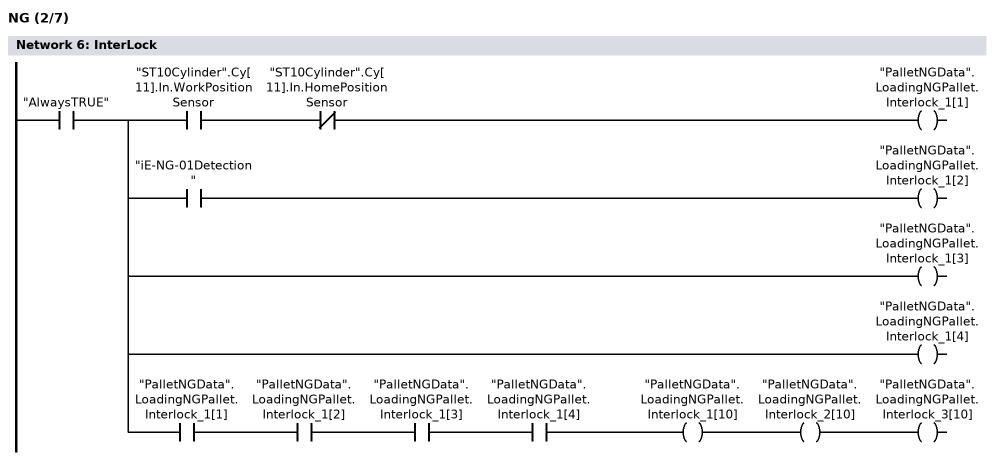
   RUNG wire#powerrail
      Contact( "AlwaysTRUE" )
      wire#w1
      Contact( "ST10Cylinder".Cy[11].In.WorkPositionSensor )
      I_Contact( "ST10Cylinder".Cy[11].In.HomePositionSensor )
      Coil( "PalletNGData".LoadingNGPallet.Interlock_1[1] )
   END_RUNG
   RUNG wire#w1
      Contact( "iE-NG-01Detection" )
      Coil( "PalletNGData".LoadingNGPallet.Interlock_1[2] )
   END_RUNG
   RUNG wire#w1
      Coil( "PalletNGData".LoadingNGPallet.Interlock_1[3] )
   END_RUNG
   RUNG wire#w1
      Coil( "PalletNGData".LoadingNGPallet.Interlock_1[4] )
   END_RUNG
   RUNG wire#w1
      Contact( "PalletNGData".LoadingNGPallet.Interlock_1[1] )
      Contact( "PalletNGData".LoadingNGPallet.Interlock_1[2] )
      Contact( "PalletNGData".LoadingNGPallet.Interlock_1[3] )
      Contact( "PalletNGData".LoadingNGPallet.Interlock_1[4] )
      Coil( "PalletNGData".LoadingNGPallet.Interlock_1[10] )
      Coil( "PalletNGData".LoadingNGPallet.Interlock_2[10] )
      Coil( "PalletNGData".LoadingNGPallet.Interlock_3[10] )
   END_RUNG
   // the same network as SCL:
   "PalletNGData".LoadingNGPallet.Interlock_1[1] := "AlwaysTRUE" AND "ST10Cylinder".Cy[11].In.WorkPositionSensor AND NOT "ST10Cylinder".Cy[11].In.HomePositionSensor;
   "PalletNGData".LoadingNGPallet.Interlock_1[2] := "AlwaysTRUE" AND "iE-NG-01Detection";
   "PalletNGData".LoadingNGPallet.Interlock_1[3] := "AlwaysTRUE";
   "PalletNGData".LoadingNGPallet.Interlock_1[4] := "AlwaysTRUE";
   #_w1 := "AlwaysTRUE" AND "PalletNGData".LoadingNGPallet.Interlock_1[1] AND "PalletNGData".LoadingNGPallet.Interlock_1[2] AND "PalletNGData".LoadingNGPallet.Interlock_1[3] AND "PalletNGData".LoadingNGPallet.Interlock_1[4];
   "PalletNGData".LoadingNGPallet.Interlock_1[10] := #_w1;
   "PalletNGData".LoadingNGPallet.Interlock_2[10] := #_w1;
   "PalletNGData".LoadingNGPallet.Interlock_3[10] := #_w1;
END_REGION

REGION Network 7: NG_Button
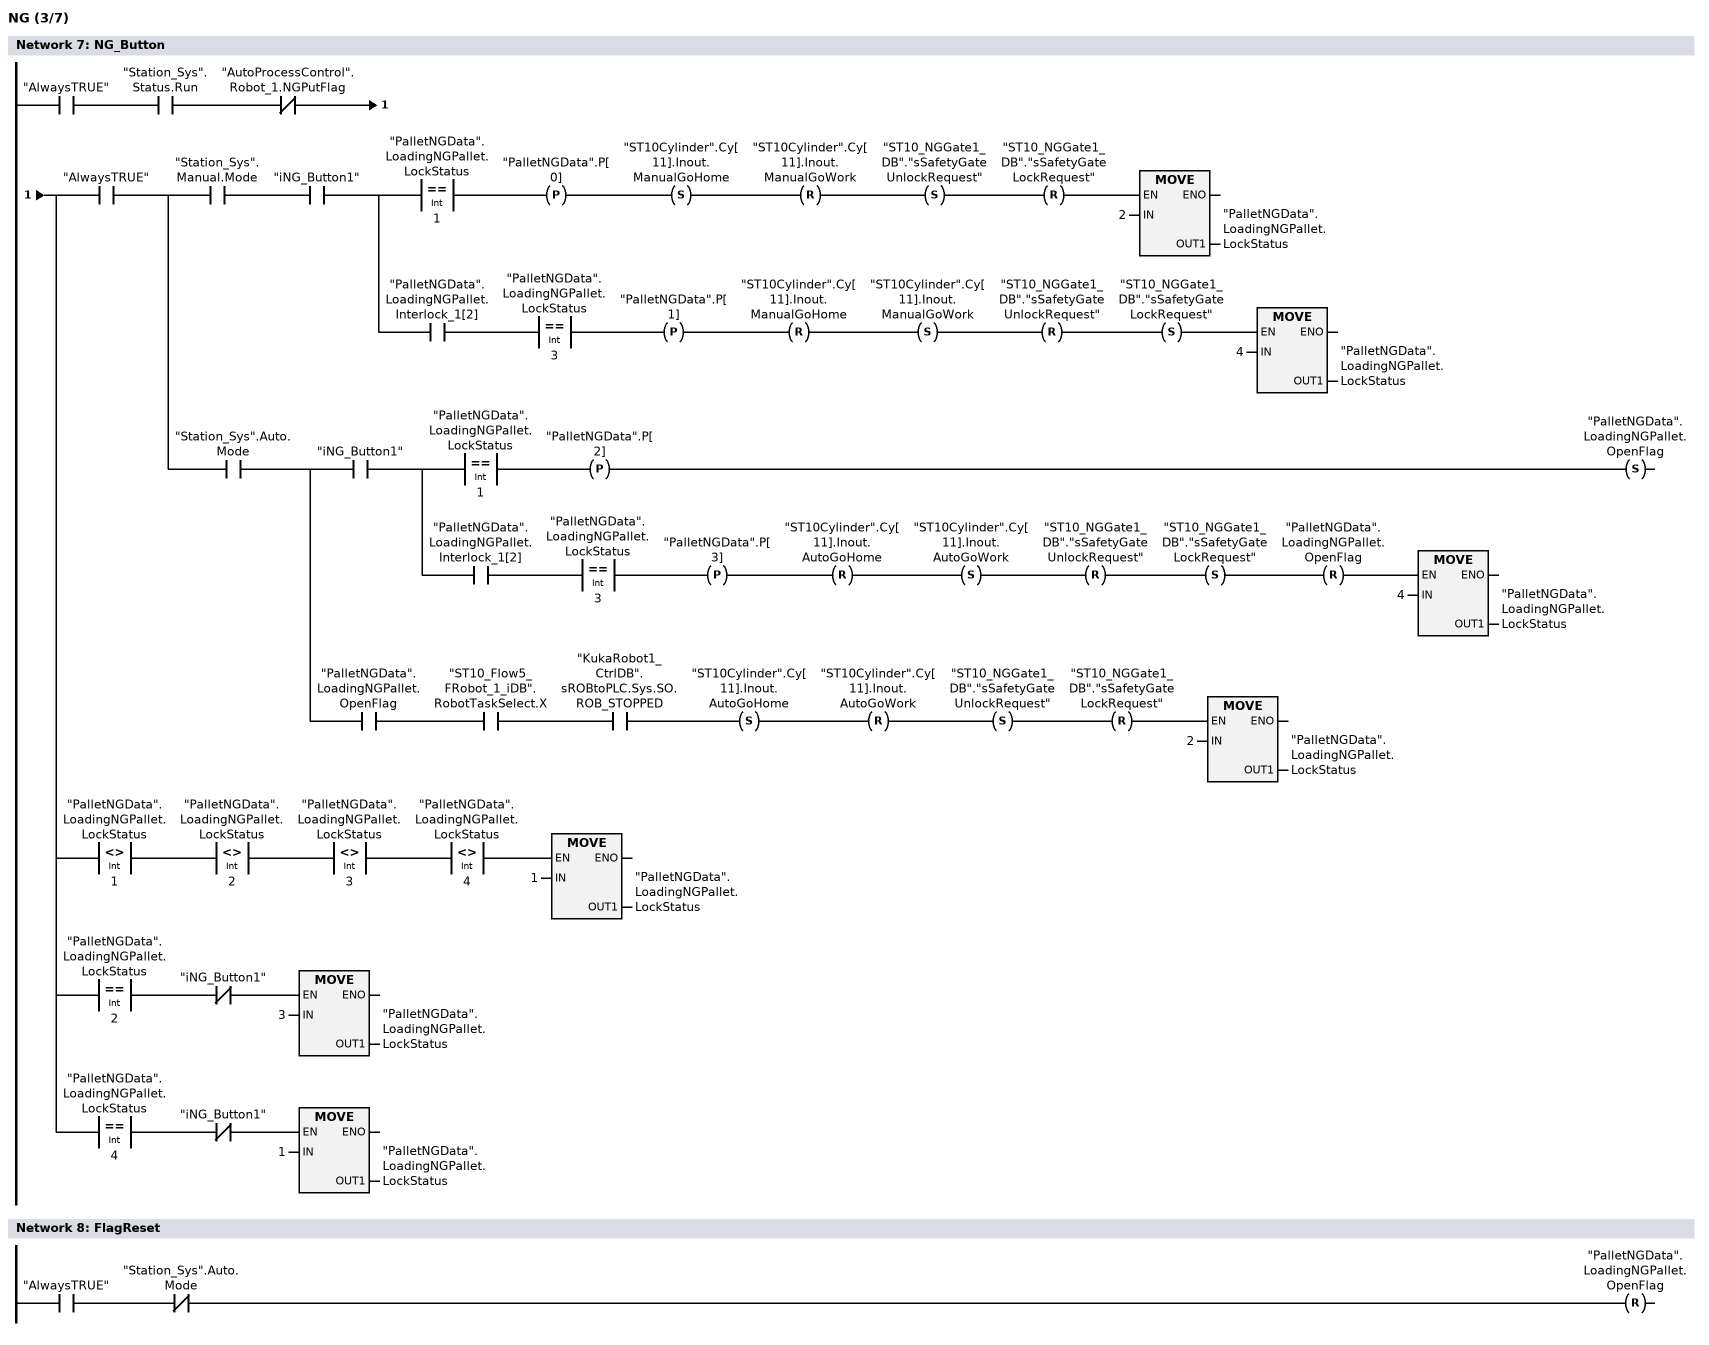
   RUNG wire#powerrail
      Contact( "AlwaysTRUE" )
      Contact( "Station_Sys".Status.Run )
      I_Contact( "AutoProcessControl".Robot_1.NGPutFlag )
      wire#w1
      Contact( "AlwaysTRUE" )
      wire#w2
      Contact( "Station_Sys".Manual.Mode )
      Contact( "iNG_Button1" )
      wire#w3
      { S7_Templates := "SrcType := Int" } EQ_Contact(in1 := "PalletNGData".LoadingNGPallet.LockStatus, in2 := 1)
      P_Trig( "PalletNGData".P[0] )
      S_Coil( "ST10Cylinder".Cy[11].Inout.ManualGoHome )
      R_Coil( "ST10Cylinder".Cy[11].Inout.ManualGoWork )
      S_Coil( "ST10_NGGate1_DB"."sSafetyGate UnlockRequest" )
      R_Coil( "ST10_NGGate1_DB"."sSafetyGate LockRequest" )
      Move(in := 2, out1 => "PalletNGData".LoadingNGPallet.LockStatus)
   END_RUNG
   RUNG wire#w3
      Contact( "PalletNGData".LoadingNGPallet.Interlock_1[2] )
      { S7_Templates := "SrcType := Int" } EQ_Contact(in1 := "PalletNGData".LoadingNGPallet.LockStatus, in2 := 3)
      P_Trig( "PalletNGData".P[1] )
      R_Coil( "ST10Cylinder".Cy[11].Inout.ManualGoHome )
      S_Coil( "ST10Cylinder".Cy[11].Inout.ManualGoWork )
      R_Coil( "ST10_NGGate1_DB"."sSafetyGate UnlockRequest" )
      S_Coil( "ST10_NGGate1_DB"."sSafetyGate LockRequest" )
      Move(in := 4, out1 => "PalletNGData".LoadingNGPallet.LockStatus)
   END_RUNG
   RUNG wire#w2
      Contact( "Station_Sys".Auto.Mode )
      wire#w4
      Contact( "iNG_Button1" )
      wire#w5
      { S7_Templates := "SrcType := Int" } EQ_Contact(in1 := "PalletNGData".LoadingNGPallet.LockStatus, in2 := 1)
      P_Trig( "PalletNGData".P[2] )
      S_Coil( "PalletNGData".LoadingNGPallet.OpenFlag )
   END_RUNG
   RUNG wire#w5
      Contact( "PalletNGData".LoadingNGPallet.Interlock_1[2] )
      { S7_Templates := "SrcType := Int" } EQ_Contact(in1 := "PalletNGData".LoadingNGPallet.LockStatus, in2 := 3)
      P_Trig( "PalletNGData".P[3] )
      R_Coil( "ST10Cylinder".Cy[11].Inout.AutoGoHome )
      S_Coil( "ST10Cylinder".Cy[11].Inout.AutoGoWork )
      R_Coil( "ST10_NGGate1_DB"."sSafetyGate UnlockRequest" )
      S_Coil( "ST10_NGGate1_DB"."sSafetyGate LockRequest" )
      R_Coil( "PalletNGData".LoadingNGPallet.OpenFlag )
      Move(in := 4, out1 => "PalletNGData".LoadingNGPallet.LockStatus)
   END_RUNG
   RUNG wire#w4
      Contact( "PalletNGData".LoadingNGPallet.OpenFlag )
      Contact( "ST10_Flow5_FRobot_1_iDB".RobotTaskSelect.X )
      Contact( "KukaRobot1_CtrlDB".sROBtoPLC.Sys.SO.ROB_STOPPED )
      S_Coil( "ST10Cylinder".Cy[11].Inout.AutoGoHome )
      R_Coil( "ST10Cylinder".Cy[11].Inout.AutoGoWork )
      S_Coil( "ST10_NGGate1_DB"."sSafetyGate UnlockRequest" )
      R_Coil( "ST10_NGGate1_DB"."sSafetyGate LockRequest" )
      Move(in := 2, out1 => "PalletNGData".LoadingNGPallet.LockStatus)
   END_RUNG
   RUNG wire#w1
      { S7_Templates := "SrcType := Int" } NE_Contact(in1 := "PalletNGData".LoadingNGPallet.LockStatus, in2 := 1)
      { S7_Templates := "SrcType := Int" } NE_Contact(in1 := "PalletNGData".LoadingNGPallet.LockStatus, in2 := 2)
      { S7_Templates := "SrcType := Int" } NE_Contact(in1 := "PalletNGData".LoadingNGPallet.LockStatus, in2 := 3)
      { S7_Templates := "SrcType := Int" } NE_Contact(in1 := "PalletNGData".LoadingNGPallet.LockStatus, in2 := 4)
      Move(in := 1, out1 => "PalletNGData".LoadingNGPallet.LockStatus)
   END_RUNG
   RUNG wire#w1
      { S7_Templates := "SrcType := Int" } EQ_Contact(in1 := "PalletNGData".LoadingNGPallet.LockStatus, in2 := 2)
      I_Contact( "iNG_Button1" )
      Move(in := 3, out1 => "PalletNGData".LoadingNGPallet.LockStatus)
   END_RUNG
   RUNG wire#w1
      { S7_Templates := "SrcType := Int" } EQ_Contact(in1 := "PalletNGData".LoadingNGPallet.LockStatus, in2 := 4)
      I_Contact( "iNG_Button1" )
      Move(in := 1, out1 => "PalletNGData".LoadingNGPallet.LockStatus)
   END_RUNG
   // the same network as SCL:
   #_w1 := "AlwaysTRUE" AND "Station_Sys".Status.Run AND NOT "AutoProcessControl".Robot_1.NGPutFlag;
   #_w2 := #_w1 AND "AlwaysTRUE";
   #_w3 := #_w2 AND "Station_Sys".Manual.Mode AND "iNG_Button1";
   #_w4 := #_w3 AND ("PalletNGData".LoadingNGPallet.LockStatus = 1);
   #_w5 := #_w4 AND NOT "PalletNGData".P[0];   // rising edge
   "PalletNGData".P[0] := #_w4;
   IF #_w5 THEN
       "ST10Cylinder".Cy[11].Inout.ManualGoHome := TRUE;
       "ST10Cylinder".Cy[11].Inout.ManualGoWork := FALSE;
       "ST10_NGGate1_DB"."sSafetyGate UnlockRequest" := TRUE;
       "ST10_NGGate1_DB"."sSafetyGate LockRequest" := FALSE;
       "PalletNGData".LoadingNGPallet.LockStatus := 2;
   END_IF;
   #_w6 := #_w3 AND "PalletNGData".LoadingNGPallet.Interlock_1[2] AND ("PalletNGData".LoadingNGPallet.LockStatus = 3);
   #_w7 := #_w6 AND NOT "PalletNGData".P[1];   // rising edge
   "PalletNGData".P[1] := #_w6;
   IF #_w7 THEN
       "ST10Cylinder".Cy[11].Inout.ManualGoHome := FALSE;
       "ST10Cylinder".Cy[11].Inout.ManualGoWork := TRUE;
       "ST10_NGGate1_DB"."sSafetyGate UnlockRequest" := FALSE;
       "ST10_NGGate1_DB"."sSafetyGate LockRequest" := TRUE;
       "PalletNGData".LoadingNGPallet.LockStatus := 4;
   END_IF;
   #_w8 := #_w2 AND "Station_Sys".Auto.Mode;
   #_w9 := #_w8 AND "iNG_Button1";
   #_w10 := #_w9 AND ("PalletNGData".LoadingNGPallet.LockStatus = 1);
   #_w11 := #_w10 AND NOT "PalletNGData".P[2];   // rising edge
   "PalletNGData".P[2] := #_w10;
   IF #_w11 THEN "PalletNGData".LoadingNGPallet.OpenFlag := TRUE; END_IF;
   #_w12 := #_w9 AND "PalletNGData".LoadingNGPallet.Interlock_1[2] AND ("PalletNGData".LoadingNGPallet.LockStatus = 3);
   #_w13 := #_w12 AND NOT "PalletNGData".P[3];   // rising edge
   "PalletNGData".P[3] := #_w12;
   IF #_w13 THEN
       "ST10Cylinder".Cy[11].Inout.AutoGoHome := FALSE;
       "ST10Cylinder".Cy[11].Inout.AutoGoWork := TRUE;
       "ST10_NGGate1_DB"."sSafetyGate UnlockRequest" := FALSE;
       "ST10_NGGate1_DB"."sSafetyGate LockRequest" := TRUE;
       "PalletNGData".LoadingNGPallet.OpenFlag := FALSE;
       "PalletNGData".LoadingNGPallet.LockStatus := 4;
   END_IF;
   IF #_w8 AND "PalletNGData".LoadingNGPallet.OpenFlag AND "ST10_Flow5_FRobot_1_iDB".RobotTaskSelect.X AND "KukaRobot1_CtrlDB".sROBtoPLC.Sys.SO.ROB_STOPPED THEN
       "ST10Cylinder".Cy[11].Inout.AutoGoHome := TRUE;
       "ST10Cylinder".Cy[11].Inout.AutoGoWork := FALSE;
       "ST10_NGGate1_DB"."sSafetyGate UnlockRequest" := TRUE;
       "ST10_NGGate1_DB"."sSafetyGate LockRequest" := FALSE;
       "PalletNGData".LoadingNGPallet.LockStatus := 2;
   END_IF;
   IF #_w1 AND ("PalletNGData".LoadingNGPallet.LockStatus <> 1) AND ("PalletNGData".LoadingNGPallet.LockStatus <> 2) AND ("PalletNGData".LoadingNGPallet.LockStatus <> 3) AND ("PalletNGData".LoadingNGPallet.LockStatus <> 4) THEN
       "PalletNGData".LoadingNGPallet.LockStatus := 1;
   END_IF;
   IF #_w1 AND ("PalletNGData".LoadingNGPallet.LockStatus = 2) AND NOT "iNG_Button1" THEN
       "PalletNGData".LoadingNGPallet.LockStatus := 3;
   END_IF;
   IF #_w1 AND ("PalletNGData".LoadingNGPallet.LockStatus = 4) AND NOT "iNG_Button1" THEN
       "PalletNGData".LoadingNGPallet.LockStatus := 1;
   END_IF;
END_REGION

REGION Network 8: FlagReset
   RUNG wire#powerrail
      Contact( "AlwaysTRUE" )
      I_Contact( "Station_Sys".Auto.Mode )
      R_Coil( "PalletNGData".LoadingNGPallet.OpenFlag )
   END_RUNG
   // the same network as SCL:
   IF "AlwaysTRUE" AND NOT "Station_Sys".Auto.Mode THEN
       "PalletNGData".LoadingNGPallet.OpenFlag := FALSE;
   END_IF;
END_REGION

REGION Network 9: NG Door
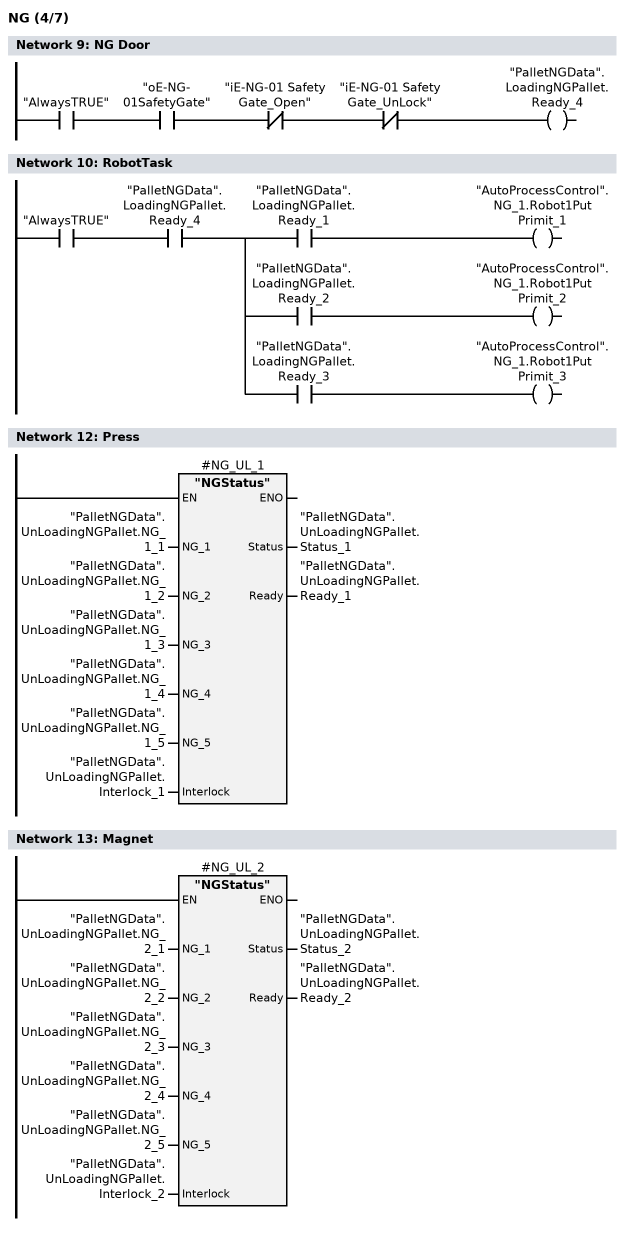
   RUNG wire#powerrail
      Contact( "AlwaysTRUE" )
      Contact( "oE-NG-01SafetyGate" )
      I_Contact( "iE-NG-01 Safety Gate_Open" )
      I_Contact( "iE-NG-01 Safety Gate_UnLock" )
      Coil( "PalletNGData".LoadingNGPallet.Ready_4 )
   END_RUNG
   // the same network as SCL:
   "PalletNGData".LoadingNGPallet.Ready_4 := "AlwaysTRUE" AND "oE-NG-01SafetyGate" AND NOT "iE-NG-01 Safety Gate_Open" AND NOT "iE-NG-01 Safety Gate_UnLock";
END_REGION

REGION Network 10: RobotTask
   RUNG wire#powerrail
      Contact( "AlwaysTRUE" )
      Contact( "PalletNGData".LoadingNGPallet.Ready_4 )
      wire#w1
      Contact( "PalletNGData".LoadingNGPallet.Ready_1 )
      Coil( "AutoProcessControl".NG_1.Robot1PutPrimit_1 )
   END_RUNG
   RUNG wire#w1
      Contact( "PalletNGData".LoadingNGPallet.Ready_2 )
      Coil( "AutoProcessControl".NG_1.Robot1PutPrimit_2 )
   END_RUNG
   RUNG wire#w1
      Contact( "PalletNGData".LoadingNGPallet.Ready_3 )
      Coil( "AutoProcessControl".NG_1.Robot1PutPrimit_3 )
   END_RUNG
   // the same network as SCL:
   #_w1 := "AlwaysTRUE" AND "PalletNGData".LoadingNGPallet.Ready_4;
   "AutoProcessControl".NG_1.Robot1PutPrimit_1 := #_w1 AND "PalletNGData".LoadingNGPallet.Ready_1;
   "AutoProcessControl".NG_1.Robot1PutPrimit_2 := #_w1 AND "PalletNGData".LoadingNGPallet.Ready_2;
   "AutoProcessControl".NG_1.Robot1PutPrimit_3 := #_w1 AND "PalletNGData".LoadingNGPallet.Ready_3;
END_REGION

REGION Network 11: --------------------------------------- UnLoad -------------------------------------------------------
END_REGION

REGION Network 12: Press
   RUNG wire#powerrail
      #NG_UL_1(NG_1 := "PalletNGData".UnLoadingNGPallet.NG_1_1, NG_2 := "PalletNGData".UnLoadingNGPallet.NG_1_2, NG_3 := "PalletNGData".UnLoadingNGPallet.NG_1_3, NG_4 := "PalletNGData".UnLoadingNGPallet.NG_1_4, NG_5 := "PalletNGData".UnLoadingNGPallet.NG_1_5, Interlock := "PalletNGData".UnLoadingNGPallet.Interlock_1, Status => "PalletNGData".UnLoadingNGPallet.Status_1, Ready => "PalletNGData".UnLoadingNGPallet.Ready_1)
   END_RUNG
   // the same network as SCL:
   #NG_UL_1(NG_1 := "PalletNGData".UnLoadingNGPallet.NG_1_1,   // "NGStatus"
            NG_2 := "PalletNGData".UnLoadingNGPallet.NG_1_2,
            NG_3 := "PalletNGData".UnLoadingNGPallet.NG_1_3,
            NG_4 := "PalletNGData".UnLoadingNGPallet.NG_1_4,
            NG_5 := "PalletNGData".UnLoadingNGPallet.NG_1_5,
            Interlock := "PalletNGData".UnLoadingNGPallet.Interlock_1,
            Status => "PalletNGData".UnLoadingNGPallet.Status_1,
            Ready => "PalletNGData".UnLoadingNGPallet.Ready_1);
END_REGION

REGION Network 13: Magnet
   RUNG wire#powerrail
      #NG_UL_2(NG_1 := "PalletNGData".UnLoadingNGPallet.NG_2_1, NG_2 := "PalletNGData".UnLoadingNGPallet.NG_2_2, NG_3 := "PalletNGData".UnLoadingNGPallet.NG_2_3, NG_4 := "PalletNGData".UnLoadingNGPallet.NG_2_4, NG_5 := "PalletNGData".UnLoadingNGPallet.NG_2_5, Interlock := "PalletNGData".UnLoadingNGPallet.Interlock_2, Status => "PalletNGData".UnLoadingNGPallet.Status_2, Ready => "PalletNGData".UnLoadingNGPallet.Ready_2)
   END_RUNG
   // the same network as SCL:
   #NG_UL_2(NG_1 := "PalletNGData".UnLoadingNGPallet.NG_2_1,   // "NGStatus"
            NG_2 := "PalletNGData".UnLoadingNGPallet.NG_2_2,
            NG_3 := "PalletNGData".UnLoadingNGPallet.NG_2_3,
            NG_4 := "PalletNGData".UnLoadingNGPallet.NG_2_4,
            NG_5 := "PalletNGData".UnLoadingNGPallet.NG_2_5,
            Interlock := "PalletNGData".UnLoadingNGPallet.Interlock_2,
            Status => "PalletNGData".UnLoadingNGPallet.Status_2,
            Ready => "PalletNGData".UnLoadingNGPallet.Ready_2);
END_REGION

REGION Network 14: Ring
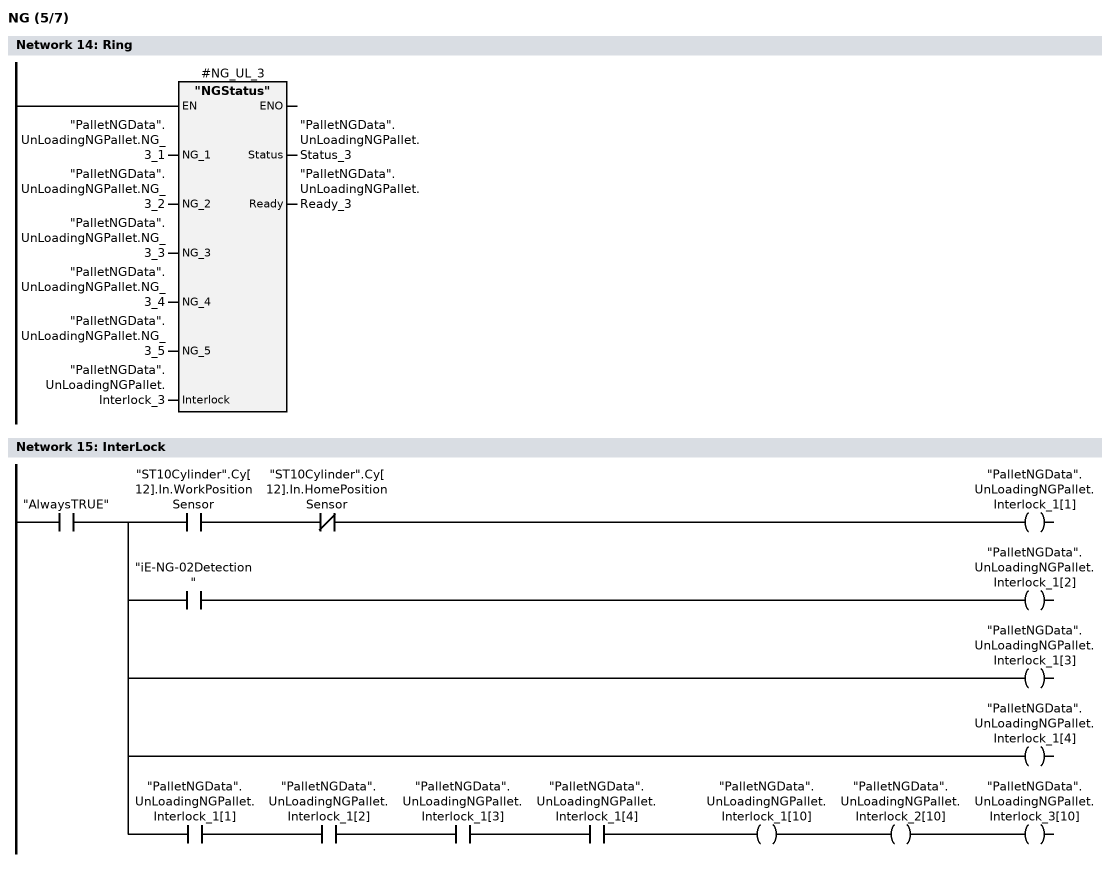
   RUNG wire#powerrail
      #NG_UL_3(NG_1 := "PalletNGData".UnLoadingNGPallet.NG_3_1, NG_2 := "PalletNGData".UnLoadingNGPallet.NG_3_2, NG_3 := "PalletNGData".UnLoadingNGPallet.NG_3_3, NG_4 := "PalletNGData".UnLoadingNGPallet.NG_3_4, NG_5 := "PalletNGData".UnLoadingNGPallet.NG_3_5, Interlock := "PalletNGData".UnLoadingNGPallet.Interlock_3, Status => "PalletNGData".UnLoadingNGPallet.Status_3, Ready => "PalletNGData".UnLoadingNGPallet.Ready_3)
   END_RUNG
   // the same network as SCL:
   #NG_UL_3(NG_1 := "PalletNGData".UnLoadingNGPallet.NG_3_1,   // "NGStatus"
            NG_2 := "PalletNGData".UnLoadingNGPallet.NG_3_2,
            NG_3 := "PalletNGData".UnLoadingNGPallet.NG_3_3,
            NG_4 := "PalletNGData".UnLoadingNGPallet.NG_3_4,
            NG_5 := "PalletNGData".UnLoadingNGPallet.NG_3_5,
            Interlock := "PalletNGData".UnLoadingNGPallet.Interlock_3,
            Status => "PalletNGData".UnLoadingNGPallet.Status_3,
            Ready => "PalletNGData".UnLoadingNGPallet.Ready_3);
END_REGION

REGION Network 15: InterLock
   RUNG wire#powerrail
      Contact( "AlwaysTRUE" )
      wire#w1
      Contact( "ST10Cylinder".Cy[12].In.WorkPositionSensor )
      I_Contact( "ST10Cylinder".Cy[12].In.HomePositionSensor )
      Coil( "PalletNGData".UnLoadingNGPallet.Interlock_1[1] )
   END_RUNG
   RUNG wire#w1
      Contact( "iE-NG-02Detection" )
      Coil( "PalletNGData".UnLoadingNGPallet.Interlock_1[2] )
   END_RUNG
   RUNG wire#w1
      Coil( "PalletNGData".UnLoadingNGPallet.Interlock_1[3] )
   END_RUNG
   RUNG wire#w1
      Coil( "PalletNGData".UnLoadingNGPallet.Interlock_1[4] )
   END_RUNG
   RUNG wire#w1
      Contact( "PalletNGData".UnLoadingNGPallet.Interlock_1[1] )
      Contact( "PalletNGData".UnLoadingNGPallet.Interlock_1[2] )
      Contact( "PalletNGData".UnLoadingNGPallet.Interlock_1[3] )
      Contact( "PalletNGData".UnLoadingNGPallet.Interlock_1[4] )
      Coil( "PalletNGData".UnLoadingNGPallet.Interlock_1[10] )
      Coil( "PalletNGData".UnLoadingNGPallet.Interlock_2[10] )
      Coil( "PalletNGData".UnLoadingNGPallet.Interlock_3[10] )
   END_RUNG
   // the same network as SCL:
   "PalletNGData".UnLoadingNGPallet.Interlock_1[1] := "AlwaysTRUE" AND "ST10Cylinder".Cy[12].In.WorkPositionSensor AND NOT "ST10Cylinder".Cy[12].In.HomePositionSensor;
   "PalletNGData".UnLoadingNGPallet.Interlock_1[2] := "AlwaysTRUE" AND "iE-NG-02Detection";
   "PalletNGData".UnLoadingNGPallet.Interlock_1[3] := "AlwaysTRUE";
   "PalletNGData".UnLoadingNGPallet.Interlock_1[4] := "AlwaysTRUE";
   #_w1 := "AlwaysTRUE" AND "PalletNGData".UnLoadingNGPallet.Interlock_1[1] AND "PalletNGData".UnLoadingNGPallet.Interlock_1[2] AND "PalletNGData".UnLoadingNGPallet.Interlock_1[3] AND "PalletNGData".UnLoadingNGPallet.Interlock_1[4];
   "PalletNGData".UnLoadingNGPallet.Interlock_1[10] := #_w1;
   "PalletNGData".UnLoadingNGPallet.Interlock_2[10] := #_w1;
   "PalletNGData".UnLoadingNGPallet.Interlock_3[10] := #_w1;
END_REGION

REGION Network 16: NG_Button
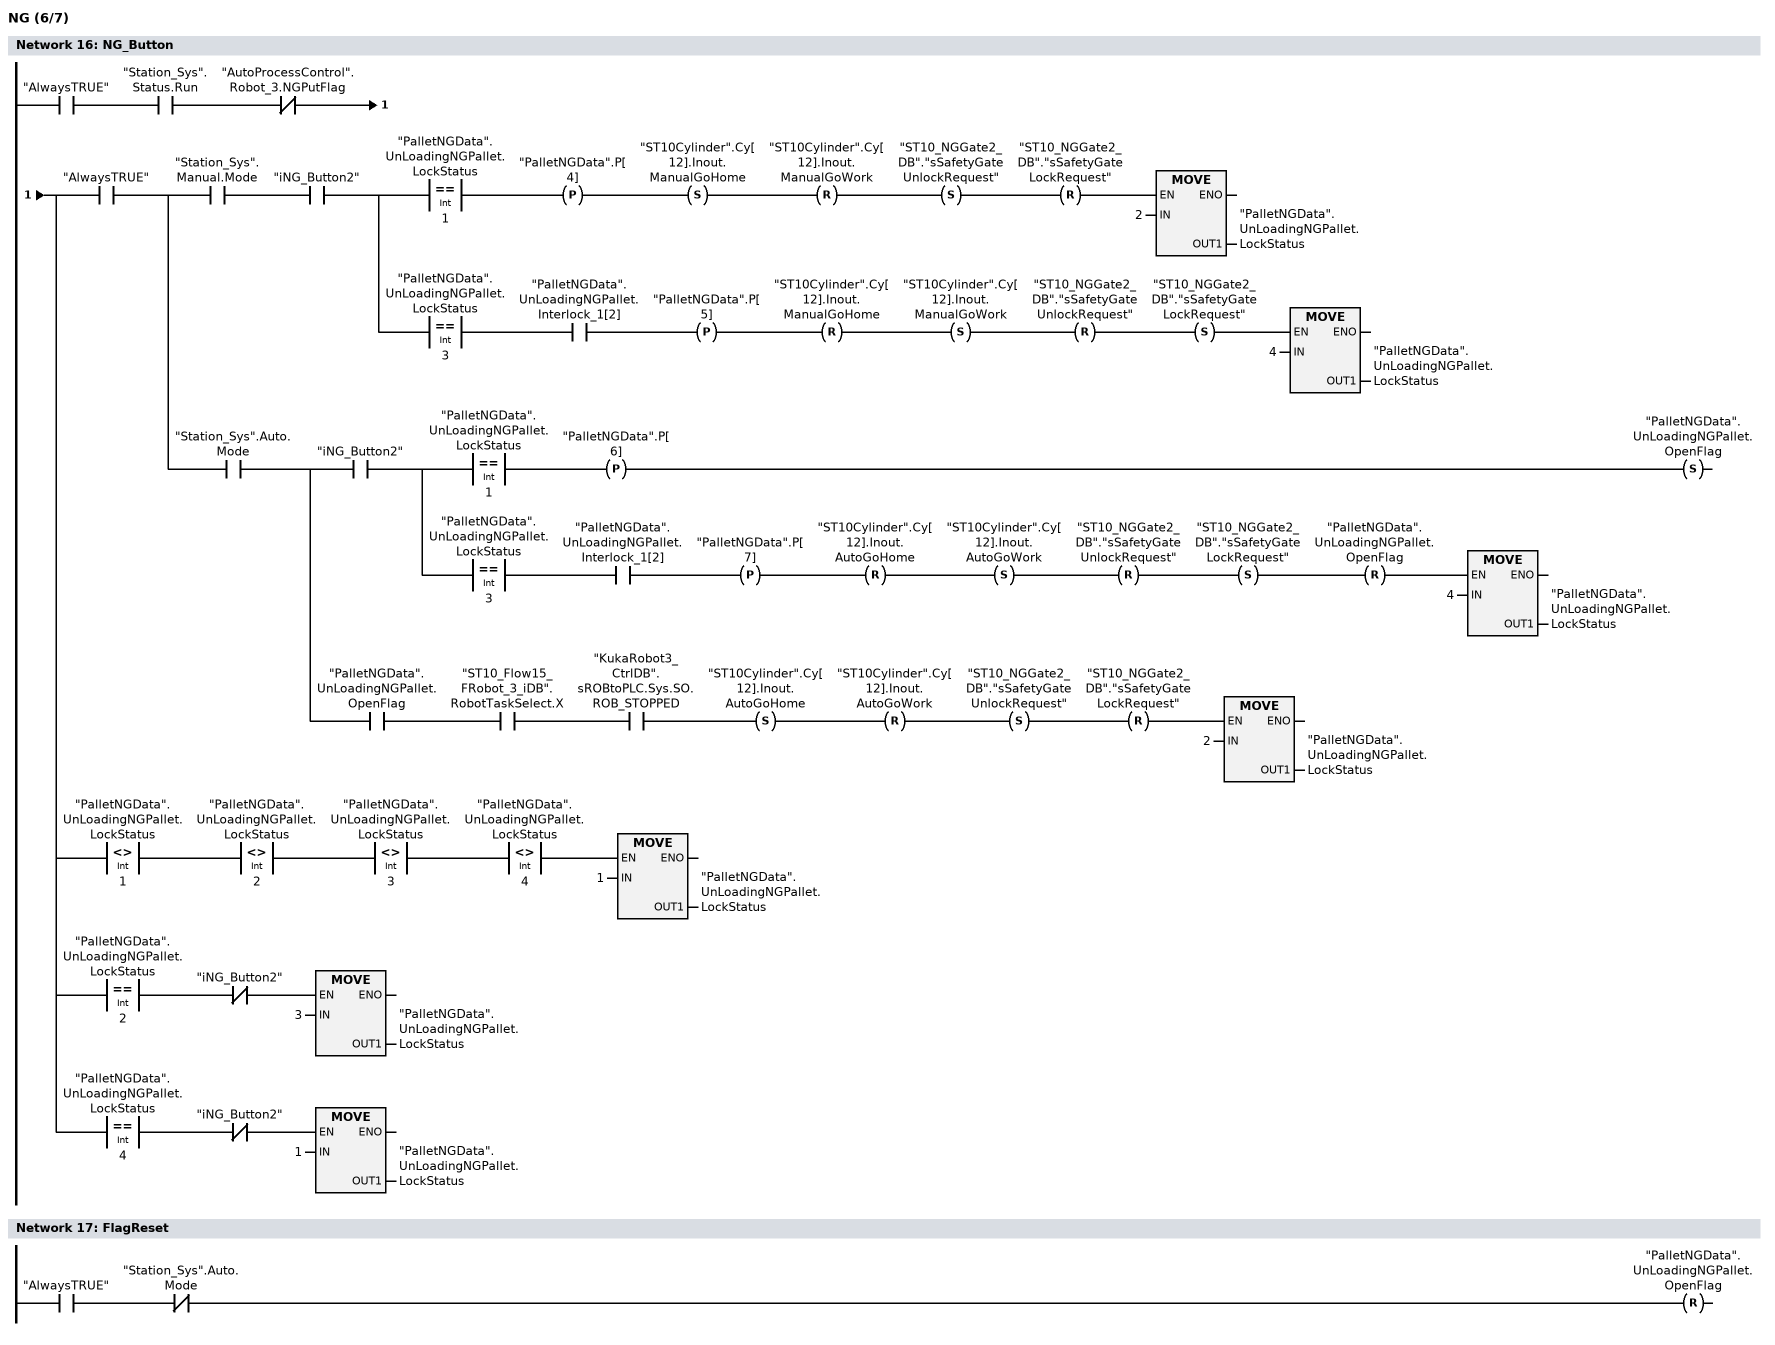
   RUNG wire#powerrail
      Contact( "AlwaysTRUE" )
      Contact( "Station_Sys".Status.Run )
      I_Contact( "AutoProcessControl".Robot_3.NGPutFlag )
      wire#w1
      Contact( "AlwaysTRUE" )
      wire#w2
      Contact( "Station_Sys".Manual.Mode )
      Contact( "iNG_Button2" )
      wire#w3
      { S7_Templates := "SrcType := Int" } EQ_Contact(in1 := "PalletNGData".UnLoadingNGPallet.LockStatus, in2 := 1)
      P_Trig( "PalletNGData".P[4] )
      S_Coil( "ST10Cylinder".Cy[12].Inout.ManualGoHome )
      R_Coil( "ST10Cylinder".Cy[12].Inout.ManualGoWork )
      S_Coil( "ST10_NGGate2_DB"."sSafetyGate UnlockRequest" )
      R_Coil( "ST10_NGGate2_DB"."sSafetyGate LockRequest" )
      Move(in := 2, out1 => "PalletNGData".UnLoadingNGPallet.LockStatus)
   END_RUNG
   RUNG wire#w3
      { S7_Templates := "SrcType := Int" } EQ_Contact(in1 := "PalletNGData".UnLoadingNGPallet.LockStatus, in2 := 3)
      Contact( "PalletNGData".UnLoadingNGPallet.Interlock_1[2] )
      P_Trig( "PalletNGData".P[5] )
      R_Coil( "ST10Cylinder".Cy[12].Inout.ManualGoHome )
      S_Coil( "ST10Cylinder".Cy[12].Inout.ManualGoWork )
      R_Coil( "ST10_NGGate2_DB"."sSafetyGate UnlockRequest" )
      S_Coil( "ST10_NGGate2_DB"."sSafetyGate LockRequest" )
      Move(in := 4, out1 => "PalletNGData".UnLoadingNGPallet.LockStatus)
   END_RUNG
   RUNG wire#w2
      Contact( "Station_Sys".Auto.Mode )
      wire#w4
      Contact( "iNG_Button2" )
      wire#w5
      { S7_Templates := "SrcType := Int" } EQ_Contact(in1 := "PalletNGData".UnLoadingNGPallet.LockStatus, in2 := 1)
      P_Trig( "PalletNGData".P[6] )
      S_Coil( "PalletNGData".UnLoadingNGPallet.OpenFlag )
   END_RUNG
   RUNG wire#w5
      { S7_Templates := "SrcType := Int" } EQ_Contact(in1 := "PalletNGData".UnLoadingNGPallet.LockStatus, in2 := 3)
      Contact( "PalletNGData".UnLoadingNGPallet.Interlock_1[2] )
      P_Trig( "PalletNGData".P[7] )
      R_Coil( "ST10Cylinder".Cy[12].Inout.AutoGoHome )
      S_Coil( "ST10Cylinder".Cy[12].Inout.AutoGoWork )
      R_Coil( "ST10_NGGate2_DB"."sSafetyGate UnlockRequest" )
      S_Coil( "ST10_NGGate2_DB"."sSafetyGate LockRequest" )
      R_Coil( "PalletNGData".UnLoadingNGPallet.OpenFlag )
      Move(in := 4, out1 => "PalletNGData".UnLoadingNGPallet.LockStatus)
   END_RUNG
   RUNG wire#w4
      Contact( "PalletNGData".UnLoadingNGPallet.OpenFlag )
      Contact( "ST10_Flow15_FRobot_3_iDB".RobotTaskSelect.X )
      Contact( "KukaRobot3_CtrlDB".sROBtoPLC.Sys.SO.ROB_STOPPED )
      S_Coil( "ST10Cylinder".Cy[12].Inout.AutoGoHome )
      R_Coil( "ST10Cylinder".Cy[12].Inout.AutoGoWork )
      S_Coil( "ST10_NGGate2_DB"."sSafetyGate UnlockRequest" )
      R_Coil( "ST10_NGGate2_DB"."sSafetyGate LockRequest" )
      Move(in := 2, out1 => "PalletNGData".UnLoadingNGPallet.LockStatus)
   END_RUNG
   RUNG wire#w1
      { S7_Templates := "SrcType := Int" } NE_Contact(in1 := "PalletNGData".UnLoadingNGPallet.LockStatus, in2 := 1)
      { S7_Templates := "SrcType := Int" } NE_Contact(in1 := "PalletNGData".UnLoadingNGPallet.LockStatus, in2 := 2)
      { S7_Templates := "SrcType := Int" } NE_Contact(in1 := "PalletNGData".UnLoadingNGPallet.LockStatus, in2 := 3)
      { S7_Templates := "SrcType := Int" } NE_Contact(in1 := "PalletNGData".UnLoadingNGPallet.LockStatus, in2 := 4)
      Move(in := 1, out1 => "PalletNGData".UnLoadingNGPallet.LockStatus)
   END_RUNG
   RUNG wire#w1
      { S7_Templates := "SrcType := Int" } EQ_Contact(in1 := "PalletNGData".UnLoadingNGPallet.LockStatus, in2 := 2)
      I_Contact( "iNG_Button2" )
      Move(in := 3, out1 => "PalletNGData".UnLoadingNGPallet.LockStatus)
   END_RUNG
   RUNG wire#w1
      { S7_Templates := "SrcType := Int" } EQ_Contact(in1 := "PalletNGData".UnLoadingNGPallet.LockStatus, in2 := 4)
      I_Contact( "iNG_Button2" )
      Move(in := 1, out1 => "PalletNGData".UnLoadingNGPallet.LockStatus)
   END_RUNG
   // the same network as SCL:
   #_w1 := "AlwaysTRUE" AND "Station_Sys".Status.Run AND NOT "AutoProcessControl".Robot_3.NGPutFlag;
   #_w2 := #_w1 AND "AlwaysTRUE";
   #_w3 := #_w2 AND "Station_Sys".Manual.Mode AND "iNG_Button2";
   #_w4 := #_w3 AND ("PalletNGData".UnLoadingNGPallet.LockStatus = 1);
   #_w5 := #_w4 AND NOT "PalletNGData".P[4];   // rising edge
   "PalletNGData".P[4] := #_w4;
   IF #_w5 THEN
       "ST10Cylinder".Cy[12].Inout.ManualGoHome := TRUE;
       "ST10Cylinder".Cy[12].Inout.ManualGoWork := FALSE;
       "ST10_NGGate2_DB"."sSafetyGate UnlockRequest" := TRUE;
       "ST10_NGGate2_DB"."sSafetyGate LockRequest" := FALSE;
       "PalletNGData".UnLoadingNGPallet.LockStatus := 2;
   END_IF;
   #_w6 := #_w3 AND ("PalletNGData".UnLoadingNGPallet.LockStatus = 3) AND "PalletNGData".UnLoadingNGPallet.Interlock_1[2];
   #_w7 := #_w6 AND NOT "PalletNGData".P[5];   // rising edge
   "PalletNGData".P[5] := #_w6;
   IF #_w7 THEN
       "ST10Cylinder".Cy[12].Inout.ManualGoHome := FALSE;
       "ST10Cylinder".Cy[12].Inout.ManualGoWork := TRUE;
       "ST10_NGGate2_DB"."sSafetyGate UnlockRequest" := FALSE;
       "ST10_NGGate2_DB"."sSafetyGate LockRequest" := TRUE;
       "PalletNGData".UnLoadingNGPallet.LockStatus := 4;
   END_IF;
   #_w8 := #_w2 AND "Station_Sys".Auto.Mode;
   #_w9 := #_w8 AND "iNG_Button2";
   #_w10 := #_w9 AND ("PalletNGData".UnLoadingNGPallet.LockStatus = 1);
   #_w11 := #_w10 AND NOT "PalletNGData".P[6];   // rising edge
   "PalletNGData".P[6] := #_w10;
   IF #_w11 THEN "PalletNGData".UnLoadingNGPallet.OpenFlag := TRUE; END_IF;
   #_w12 := #_w9 AND ("PalletNGData".UnLoadingNGPallet.LockStatus = 3) AND "PalletNGData".UnLoadingNGPallet.Interlock_1[2];
   #_w13 := #_w12 AND NOT "PalletNGData".P[7];   // rising edge
   "PalletNGData".P[7] := #_w12;
   IF #_w13 THEN
       "ST10Cylinder".Cy[12].Inout.AutoGoHome := FALSE;
       "ST10Cylinder".Cy[12].Inout.AutoGoWork := TRUE;
       "ST10_NGGate2_DB"."sSafetyGate UnlockRequest" := FALSE;
       "ST10_NGGate2_DB"."sSafetyGate LockRequest" := TRUE;
       "PalletNGData".UnLoadingNGPallet.OpenFlag := FALSE;
       "PalletNGData".UnLoadingNGPallet.LockStatus := 4;
   END_IF;
   IF #_w8 AND "PalletNGData".UnLoadingNGPallet.OpenFlag AND "ST10_Flow15_FRobot_3_iDB".RobotTaskSelect.X AND "KukaRobot3_CtrlDB".sROBtoPLC.Sys.SO.ROB_STOPPED THEN
       "ST10Cylinder".Cy[12].Inout.AutoGoHome := TRUE;
       "ST10Cylinder".Cy[12].Inout.AutoGoWork := FALSE;
       "ST10_NGGate2_DB"."sSafetyGate UnlockRequest" := TRUE;
       "ST10_NGGate2_DB"."sSafetyGate LockRequest" := FALSE;
       "PalletNGData".UnLoadingNGPallet.LockStatus := 2;
   END_IF;
   IF #_w1 AND ("PalletNGData".UnLoadingNGPallet.LockStatus <> 1) AND ("PalletNGData".UnLoadingNGPallet.LockStatus <> 2) AND ("PalletNGData".UnLoadingNGPallet.LockStatus <> 3) AND ("PalletNGData".UnLoadingNGPallet.LockStatus <> 4) THEN
       "PalletNGData".UnLoadingNGPallet.LockStatus := 1;
   END_IF;
   IF #_w1 AND ("PalletNGData".UnLoadingNGPallet.LockStatus = 2) AND NOT "iNG_Button2" THEN
       "PalletNGData".UnLoadingNGPallet.LockStatus := 3;
   END_IF;
   IF #_w1 AND ("PalletNGData".UnLoadingNGPallet.LockStatus = 4) AND NOT "iNG_Button2" THEN
       "PalletNGData".UnLoadingNGPallet.LockStatus := 1;
   END_IF;
END_REGION

REGION Network 17: FlagReset
   RUNG wire#powerrail
      Contact( "AlwaysTRUE" )
      I_Contact( "Station_Sys".Auto.Mode )
      R_Coil( "PalletNGData".UnLoadingNGPallet.OpenFlag )
   END_RUNG
   // the same network as SCL:
   IF "AlwaysTRUE" AND NOT "Station_Sys".Auto.Mode THEN
       "PalletNGData".UnLoadingNGPallet.OpenFlag := FALSE;
   END_IF;
END_REGION

REGION Network 18: NG Door
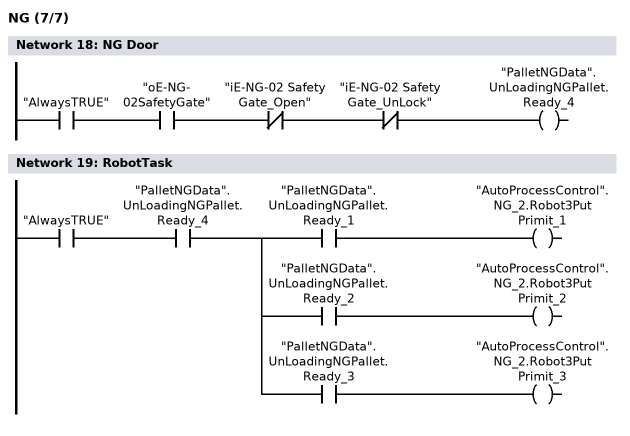
   RUNG wire#powerrail
      Contact( "AlwaysTRUE" )
      Contact( "oE-NG-02SafetyGate" )
      I_Contact( "iE-NG-02 Safety Gate_Open" )
      I_Contact( "iE-NG-02 Safety Gate_UnLock" )
      Coil( "PalletNGData".UnLoadingNGPallet.Ready_4 )
   END_RUNG
   // the same network as SCL:
   "PalletNGData".UnLoadingNGPallet.Ready_4 := "AlwaysTRUE" AND "oE-NG-02SafetyGate" AND NOT "iE-NG-02 Safety Gate_Open" AND NOT "iE-NG-02 Safety Gate_UnLock";
END_REGION

REGION Network 19: RobotTask
   RUNG wire#powerrail
      Contact( "AlwaysTRUE" )
      Contact( "PalletNGData".UnLoadingNGPallet.Ready_4 )
      wire#w1
      Contact( "PalletNGData".UnLoadingNGPallet.Ready_1 )
      Coil( "AutoProcessControl".NG_2.Robot3PutPrimit_1 )
   END_RUNG
   RUNG wire#w1
      Contact( "PalletNGData".UnLoadingNGPallet.Ready_2 )
      Coil( "AutoProcessControl".NG_2.Robot3PutPrimit_2 )
   END_RUNG
   RUNG wire#w1
      Contact( "PalletNGData".UnLoadingNGPallet.Ready_3 )
      Coil( "AutoProcessControl".NG_2.Robot3PutPrimit_3 )
   END_RUNG
   // the same network as SCL:
   #_w1 := "AlwaysTRUE" AND "PalletNGData".UnLoadingNGPallet.Ready_4;
   "AutoProcessControl".NG_2.Robot3PutPrimit_1 := #_w1 AND "PalletNGData".UnLoadingNGPallet.Ready_1;
   "AutoProcessControl".NG_2.Robot3PutPrimit_2 := #_w1 AND "PalletNGData".UnLoadingNGPallet.Ready_2;
   "AutoProcessControl".NG_2.Robot3PutPrimit_3 := #_w1 AND "PalletNGData".UnLoadingNGPallet.Ready_3;
END_REGION
END_FUNCTION_BLOCK

FUNCTION_BLOCK "NGStatus"   // FB2900, LAD
{ S7_Optimized_Access := 'TRUE' }
// stored: AutoNumber false, MemoryReserve 100, SetENOAutomatically false
   VAR_INPUT
      NG_1 : Bool;
      NG_2 : Bool;
      NG_3 : Bool;
      NG_4 : Bool;
      NG_5 : Bool;
   END_VAR
   VAR_OUTPUT
      Status : Int;
      Ready : Bool;
   END_VAR
   VAR_IN_OUT
      Interlock : Array[1..10] of Bool;
   END_VAR
   VAR
      AlwaysOn : Bool;
      NG_Delay : Array[1..10] of TON_TIME;
      NG_DelayTime { S7_SetPoint := 'True'} : Array[1..10] of DInt;
   END_VAR
   // NG_DelayTime[1..10] := 1000;
BEGIN

REGION Network 1: #AlwaysOn
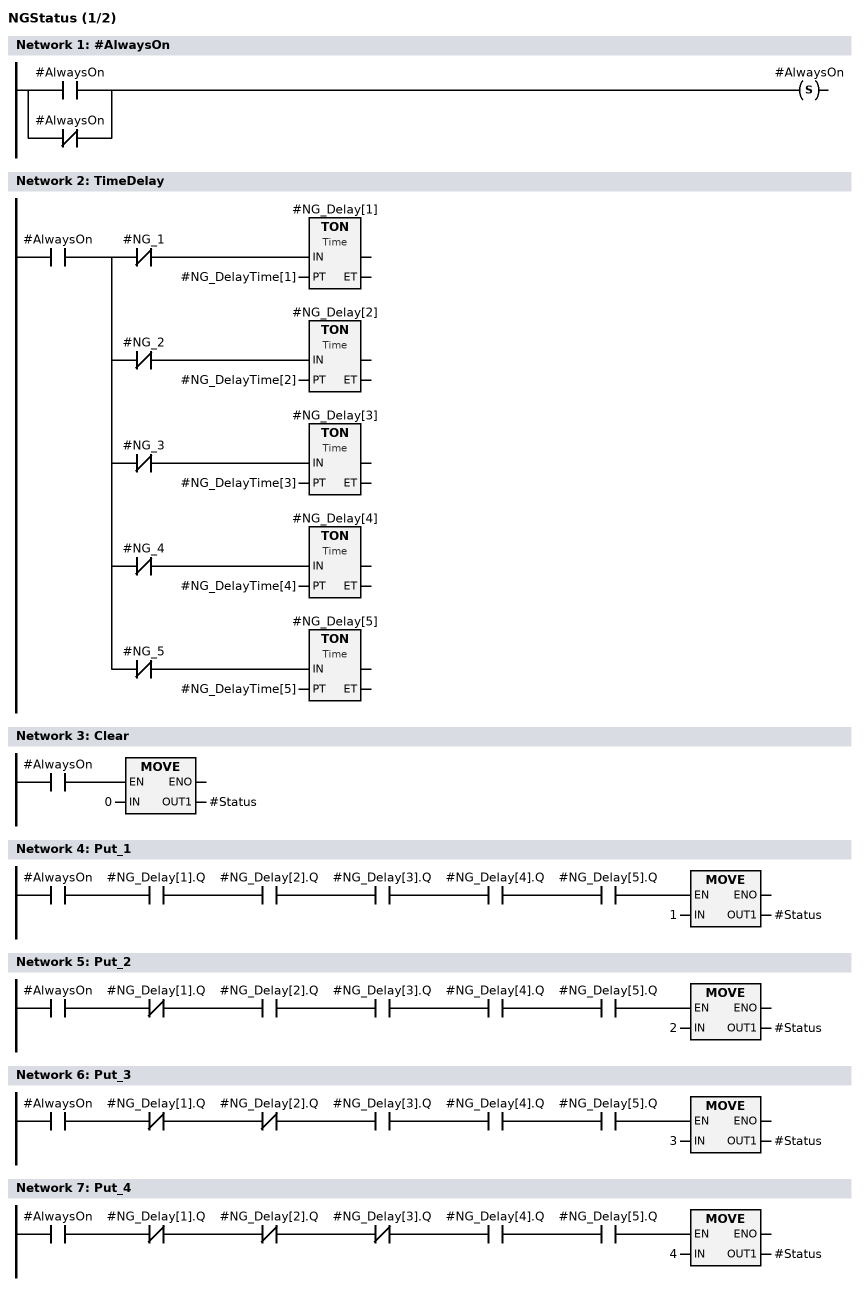
   RUNG wire#powerrail
      Contact( #AlwaysOn )
      wire#w1
      S_Coil( #AlwaysOn )
   END_RUNG
   RUNG wire#powerrail
      I_Contact( #AlwaysOn )
   END_RUNG wire#w1
   // the same network as SCL:
   IF #AlwaysOn OR NOT #AlwaysOn THEN #AlwaysOn := TRUE; END_IF;
END_REGION

REGION Network 2: TimeDelay
   RUNG wire#powerrail
      Contact( #AlwaysOn )
      wire#w1
      I_Contact( #NG_1 )
      { S7_Templates := "time_type := Time" } #NG_Delay[1].TON(pt := #NG_DelayTime[1], et =>)
   END_RUNG
   RUNG wire#w1
      I_Contact( #NG_2 )
      { S7_Templates := "time_type := Time" } #NG_Delay[2].TON(pt := #NG_DelayTime[2], et =>)
   END_RUNG
   RUNG wire#w1
      I_Contact( #NG_3 )
      { S7_Templates := "time_type := Time" } #NG_Delay[3].TON(pt := #NG_DelayTime[3], et =>)
   END_RUNG
   RUNG wire#w1
      I_Contact( #NG_4 )
      { S7_Templates := "time_type := Time" } #NG_Delay[4].TON(pt := #NG_DelayTime[4], et =>)
   END_RUNG
   RUNG wire#w1
      I_Contact( #NG_5 )
      { S7_Templates := "time_type := Time" } #NG_Delay[5].TON(pt := #NG_DelayTime[5], et =>)
   END_RUNG
   // the same network as SCL:
   #NG_Delay[1].TON(IN := #AlwaysOn AND NOT #NG_1, PT := #NG_DelayTime[1]);
   #NG_Delay[2].TON(IN := #AlwaysOn AND NOT #NG_2, PT := #NG_DelayTime[2]);
   #NG_Delay[3].TON(IN := #AlwaysOn AND NOT #NG_3, PT := #NG_DelayTime[3]);
   #NG_Delay[4].TON(IN := #AlwaysOn AND NOT #NG_4, PT := #NG_DelayTime[4]);
   #NG_Delay[5].TON(IN := #AlwaysOn AND NOT #NG_5, PT := #NG_DelayTime[5]);
END_REGION

REGION Network 3: Clear
   RUNG wire#powerrail
      Contact( #AlwaysOn )
      Move(in := 0, out1 => #Status)
   END_RUNG
   // the same network as SCL:
   IF #AlwaysOn THEN #Status := 0; END_IF;
END_REGION

REGION Network 4: Put_1
   RUNG wire#powerrail
      Contact( #AlwaysOn )
      Contact( #NG_Delay[1].Q )
      Contact( #NG_Delay[2].Q )
      Contact( #NG_Delay[3].Q )
      Contact( #NG_Delay[4].Q )
      Contact( #NG_Delay[5].Q )
      Move(in := 1, out1 => #Status)
   END_RUNG
   // the same network as SCL:
   IF #AlwaysOn AND #NG_Delay[1].Q AND #NG_Delay[2].Q AND #NG_Delay[3].Q AND #NG_Delay[4].Q AND #NG_Delay[5].Q THEN
       #Status := 1;
   END_IF;
END_REGION

REGION Network 5: Put_2
   RUNG wire#powerrail
      Contact( #AlwaysOn )
      I_Contact( #NG_Delay[1].Q )
      Contact( #NG_Delay[2].Q )
      Contact( #NG_Delay[3].Q )
      Contact( #NG_Delay[4].Q )
      Contact( #NG_Delay[5].Q )
      Move(in := 2, out1 => #Status)
   END_RUNG
   // the same network as SCL:
   IF #AlwaysOn AND NOT #NG_Delay[1].Q AND #NG_Delay[2].Q AND #NG_Delay[3].Q AND #NG_Delay[4].Q AND #NG_Delay[5].Q THEN
       #Status := 2;
   END_IF;
END_REGION

REGION Network 6: Put_3
   RUNG wire#powerrail
      Contact( #AlwaysOn )
      I_Contact( #NG_Delay[1].Q )
      I_Contact( #NG_Delay[2].Q )
      Contact( #NG_Delay[3].Q )
      Contact( #NG_Delay[4].Q )
      Contact( #NG_Delay[5].Q )
      Move(in := 3, out1 => #Status)
   END_RUNG
   // the same network as SCL:
   IF #AlwaysOn AND NOT #NG_Delay[1].Q AND NOT #NG_Delay[2].Q AND #NG_Delay[3].Q AND #NG_Delay[4].Q AND #NG_Delay[5].Q THEN
       #Status := 3;
   END_IF;
END_REGION

REGION Network 7: Put_4
   RUNG wire#powerrail
      Contact( #AlwaysOn )
      I_Contact( #NG_Delay[1].Q )
      I_Contact( #NG_Delay[2].Q )
      I_Contact( #NG_Delay[3].Q )
      Contact( #NG_Delay[4].Q )
      Contact( #NG_Delay[5].Q )
      Move(in := 4, out1 => #Status)
   END_RUNG
   // the same network as SCL:
   IF #AlwaysOn AND NOT #NG_Delay[1].Q AND NOT #NG_Delay[2].Q AND NOT #NG_Delay[3].Q AND #NG_Delay[4].Q AND #NG_Delay[5].Q THEN
       #Status := 4;
   END_IF;
END_REGION

REGION Network 8: Put_5
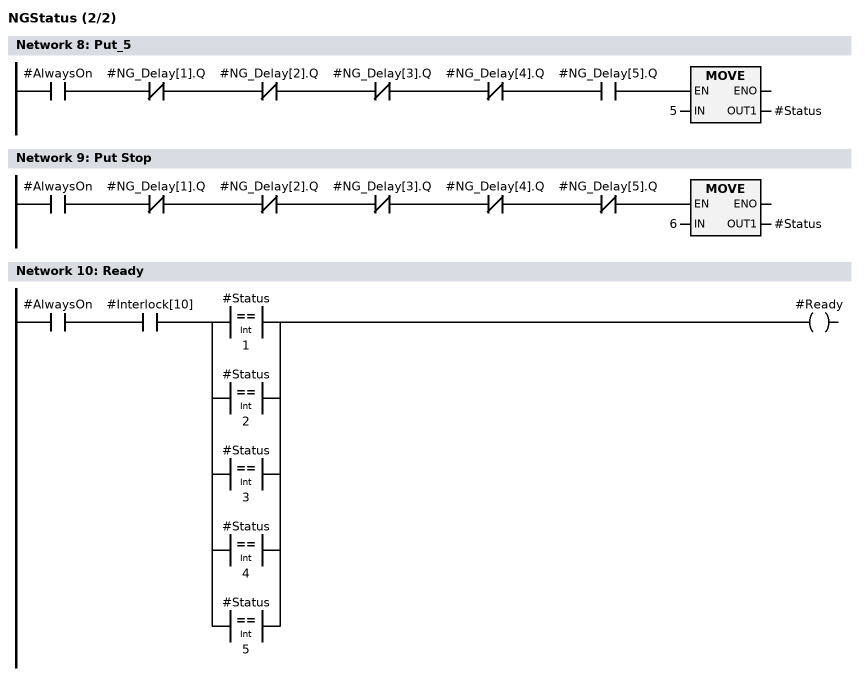
   RUNG wire#powerrail
      Contact( #AlwaysOn )
      I_Contact( #NG_Delay[1].Q )
      I_Contact( #NG_Delay[2].Q )
      I_Contact( #NG_Delay[3].Q )
      I_Contact( #NG_Delay[4].Q )
      Contact( #NG_Delay[5].Q )
      Move(in := 5, out1 => #Status)
   END_RUNG
   // the same network as SCL:
   IF #AlwaysOn AND NOT #NG_Delay[1].Q AND NOT #NG_Delay[2].Q AND NOT #NG_Delay[3].Q AND NOT #NG_Delay[4].Q AND #NG_Delay[5].Q THEN
       #Status := 5;
   END_IF;
END_REGION

REGION Network 9: Put Stop
   RUNG wire#powerrail
      Contact( #AlwaysOn )
      I_Contact( #NG_Delay[1].Q )
      I_Contact( #NG_Delay[2].Q )
      I_Contact( #NG_Delay[3].Q )
      I_Contact( #NG_Delay[4].Q )
      I_Contact( #NG_Delay[5].Q )
      Move(in := 6, out1 => #Status)
   END_RUNG
   // the same network as SCL:
   IF #AlwaysOn AND NOT #NG_Delay[1].Q AND NOT #NG_Delay[2].Q AND NOT #NG_Delay[3].Q AND NOT #NG_Delay[4].Q AND NOT #NG_Delay[5].Q THEN
       #Status := 6;
   END_IF;
END_REGION

REGION Network 10: Ready
   RUNG wire#powerrail
      Contact( #AlwaysOn )
      Contact( #Interlock[10] )
      wire#w1
      { S7_Templates := "SrcType := Int" } EQ_Contact(in1 := #Status, in2 := 1)
      wire#w2
      Coil( #Ready )
   END_RUNG
   RUNG wire#w1
      { S7_Templates := "SrcType := Int" } EQ_Contact(in1 := #Status, in2 := 2)
   END_RUNG wire#w2
   RUNG wire#w1
      { S7_Templates := "SrcType := Int" } EQ_Contact(in1 := #Status, in2 := 3)
   END_RUNG wire#w2
   RUNG wire#w1
      { S7_Templates := "SrcType := Int" } EQ_Contact(in1 := #Status, in2 := 4)
   END_RUNG wire#w2
   RUNG wire#w1
      { S7_Templates := "SrcType := Int" } EQ_Contact(in1 := #Status, in2 := 5)
   END_RUNG wire#w2
   // the same network as SCL:
   #Ready := #AlwaysOn AND #Interlock[10] AND ((#Status = 1) OR (#Status = 2) OR (#Status = 3) OR (#Status = 4) OR (#Status = 5));
END_REGION
END_FUNCTION_BLOCK

FUNCTION_BLOCK "AutoProcessDataPopUp"
{ S7_Optimized_Access := 'TRUE' }
VERSION : 0.1
   VAR_IN_OUT 
      idx { ExternalAccessible := 'False'; ExternalVisible := 'False'; ExternalWritable := 'False'} : Int;
   END_VAR

   VAR_TEMP 
      DefaultData : "ProcessData";
   END_VAR


